  MoveL 652 to (-21.11, 309.47, 290) mm, rotated rx -90 ry -25 rz -110.46 deg; joints [2.992, -46.033, 98.025, 220.576, 108.57, -187.083, -1369.544]
  MoveL 653 to (-10.16, 196.36, 0) mm, rotated rx -90 ry -25 rz 39.27 deg; joints [-7.468, -49.927, 106.451, 214.616, 108.422, -179.076, -1519.273]
  Set speed (60.0 mm/s)
  MoveL 654 to (37.62, 209.05, 0) mm, rotated rx -90 ry -25 rz 92.57 deg; joints [-7.468, -49.977, 106.447, 214.605, 108.377, -179.109, -1572.574]
  MoveL 655 to (-10.16, 196.36, 0) mm, rotated rx -90 ry -25 rz 39.27 deg; joints [-7.468, -49.927, 106.451, 214.616, 108.422, -179.076, -1519.273]
  Set speed (60.0 mm/s)
  MoveL 656 to (-5.87, 195.78, 10) mm, rotated rx -90 ry -25 rz 43.82 deg; joints [-7.088, -49.822, 106.25, 214.856, 108.462, -179.315, -1523.823]
  MoveL 657 to (-1.12, 195.49, 20) mm, rotated rx -90 ry -25 rz 48.82 deg; joints [-6.709, -49.715, 106.043, 215.095, 108.501, -179.557, -1528.824]
  MoveL 658 to (4.03, 195.62, 30) mm, rotated rx -90 ry -25 rz 54.24 deg; joints [-6.332, -49.606, 105.829, 215.332, 108.536, -179.801, -1534.238]
  MoveL 659 to (9.5, 196.25, 40) mm, rotated rx -90 ry -25 rz 60.02 deg; joints [-5.956, -49.496, 105.609, 215.565, 108.567, -180.049, -1540.02]
  MoveL 660 to (15.19, 197.47, 50) mm, rotated rx -90 ry -25 rz 66.13 deg; joints [-5.581, -49.385, 105.383, 215.797, 108.596, -180.3, -1546.127]
  MoveL 661 to (21, 199.35, 60) mm, rotated rx -90 ry -25 rz 72.51 deg; joints [-5.207, -49.274, 105.15, 216.025, 108.62, -180.554, -1552.515]
  MoveL 662 to (26.8, 201.92, 70) mm, rotated rx -90 ry -25 rz 79.14 deg; joints [-4.834, -49.162, 104.91, 216.251, 108.64, -180.811, -1559.135]
  MoveL 663 to (32.46, 205.23, 80) mm, rotated rx -90 ry -25 rz 85.94 deg; joints [-4.463, -49.05, 104.664, 216.474, 108.657, -181.073, -1565.942]
  MoveL 664 to (37.86, 209.24, 90) mm, rotated rx -90 ry -25 rz 92.89 deg; joints [-4.093, -48.937, 104.412, 216.694, 108.67, -181.338, -1572.888]
  MoveL 665 to (42.85, 213.95, 100) mm, rotated rx -90 ry -25 rz 99.93 deg; joints [-3.725, -48.823, 104.153, 216.911, 108.679, -181.606, -1579.928]
  MoveL 666 to (47.33, 219.29, 110) mm, rotated rx -90 ry -25 rz 107.02 deg; joints [-3.358, -48.708, 103.888, 217.126, 108.685, -181.879, -1587.017]
  MoveL 667 to (51.17, 225.17, 120) mm, rotated rx -90 ry -25 rz 114.11 deg; joints [-2.992, -48.592, 103.616, 217.338, 108.687, -182.154, -1594.112]
  MoveL 668 to (54.3, 231.49, 130) mm, rotated rx -90 ry -25 rz 121.17 deg; joints [-2.628, -48.474, 103.338, 217.547, 108.687, -182.432, -1601.173]
  MoveL 669 to (56.65, 238.12, 140) mm, rotated rx -90 ry -25 rz 128.16 deg; joints [-2.265, -48.354, 103.054, 217.753, 108.685, -182.713, -1608.16]
  MoveL 670 to (58.18, 244.95, 150) mm, rotated rx -90 ry -25 rz 135.04 deg; joints [-1.904, -48.231, 102.763, 217.957, 108.681, -182.996, -1615.039]
  MoveL 671 to (58.89, 251.83, 160) mm, rotated rx -90 ry -25 rz 141.78 deg; joints [-1.544, -48.104, 102.465, 218.159, 108.676, -183.281, -1621.776]
  MoveL 672 to (58.8, 258.62, 170) mm, rotated rx -90 ry -25 rz 148.34 deg; joints [-1.185, -47.974, 102.162, 218.358, 108.669, -183.568, -1628.339]
  MoveL 673 to (57.96, 265.2, 180) mm, rotated rx -90 ry -25 rz 154.7 deg; joints [-0.828, -47.839, 101.852, 218.555, 108.662, -183.856, -1634.699]
  MoveL 674 to (56.44, 271.47, 190) mm, rotated rx -90 ry -25 rz 160.83 deg; joints [-0.473, -47.7, 101.535, 218.75, 108.655, -184.145, -1640.826]
  MoveL 675 to (54.33, 277.32, 200) mm, rotated rx -90 ry -25 rz 166.69 deg; joints [-0.119, -47.555, 101.213, 218.942, 108.647, -184.435, -1646.694]
  MoveL 676 to (51.74, 282.68, 210) mm, rotated rx -90 ry -25 rz 172.28 deg; joints [0.233, -47.406, 100.884, 219.133, 108.64, -184.725, -1652.275]
  MoveL 677 to (48.8, 287.5, 220) mm, rotated rx -90 ry -25 rz 177.54 deg; joints [0.584, -47.251, 100.549, 219.321, 108.632, -185.016, -1657.543]
  MoveL 678 to (45.62, 291.76, 230) mm, rotated rx -90 ry -25 rz -177.53 deg; joints [0.933, -47.091, 100.208, 219.507, 108.625, -185.308, -1662.471]
  MoveL 679 to (42.34, 295.45, 240) mm, rotated rx -90 ry -25 rz -172.97 deg; joints [1.28, -46.926, 99.86, 219.691, 108.618, -185.601, -1667.031]
  MoveL 680 to (39.07, 298.58, 250) mm, rotated rx -90 ry -25 rz -168.8 deg; joints [1.626, -46.755, 99.506, 219.873, 108.61, -185.894, -1671.197]
  MoveL 681 to (35.92, 301.18, 260) mm, rotated rx -90 ry -25 rz -165.06 deg; joints [1.97, -46.579, 99.146, 220.053, 108.603, -186.188, -1674.94]
  MoveL 682 to (33, 303.28, 270) mm, rotated rx -90 ry -25 rz -161.77 deg; joints [2.312, -46.398, 98.779, 220.231, 108.595, -186.483, -1678.23]
  MoveL 683 to (30.4, 304.94, 280) mm, rotated rx -90 ry -25 rz -158.96 deg; joints [2.653, -46.213, 98.406, 220.406, 108.587, -186.778, -1681.04]
  MoveL 684 to (28.22, 306.19, 290) mm, rotated rx -90 ry -25 rz -156.66 deg; joints [2.992, -46.023, 98.026, 220.579, 108.578, -187.075, -1683.337]
  MoveL 685 to (-21.11, 309.47, 290) mm, rotated rx -90 ry -25 rz -110.46 deg; joints [2.992, -46.033, 98.025, 220.576, 108.57, -187.083, -1729.544]
  Set speed (60.0 mm/s)
  MoveL 686 to (-18.74, 310.33, 280) mm, rotated rx -90 ry -25 rz -112.74 deg; joints [2.653, -46.23, 98.404, 220.402, 108.573, -186.791, -1727.257]
  MoveL 687 to (-15.8, 311.23, 270) mm, rotated rx -90 ry -25 rz -115.53 deg; joints [2.312, -46.424, 98.777, 220.225, 108.574, -186.502, -1724.467]
  MoveL 688 to (-12.3, 312.09, 260) mm, rotated rx -90 ry -25 rz -118.79 deg; joints [1.97, -46.614, 99.142, 220.045, 108.574, -186.214, -1721.209]
  MoveL 689 to (-8.28, 312.8, 250) mm, rotated rx -90 ry -25 rz -122.48 deg; joints [1.626, -46.801, 99.502, 219.863, 108.572, -185.928, -1717.515]
  MoveL 690 to (-3.78, 313.26, 240) mm, rotated rx -90 ry -25 rz -126.58 deg; joints [1.28, -46.983, 99.855, 219.678, 108.569, -185.643, -1713.419]
  MoveL 691 to (1.16, 313.37, 230) mm, rotated rx -90 ry -25 rz -131.05 deg; joints [0.933, -47.161, 100.201, 219.491, 108.565, -185.36, -1708.952]
  MoveL 692 to (6.46, 313.03, 220) mm, rotated rx -90 ry -25 rz -135.85 deg; joints [0.584, -47.335, 100.541, 219.301, 108.561, -185.078, -1704.147]
  MoveL 693 to (12.04, 312.14, 210) mm, rotated rx -90 ry -25 rz -140.97 deg; joints [0.233, -47.503, 100.875, 219.11, 108.557, -184.796, -1699.032]
  MoveL 694 to (17.8, 310.63, 200) mm, rotated rx -90 ry -25 rz -146.36 deg; joints [-0.119, -47.666, 101.203, 218.916, 108.553, -184.515, -1693.638]
  MoveL 695 to (23.62, 308.44, 190) mm, rotated rx -90 ry -25 rz -152.01 deg; joints [-0.473, -47.824, 101.524, 218.721, 108.549, -184.234, -1687.993]
  MoveL 696 to (29.38, 305.54, 180) mm, rotated rx -90 ry -25 rz -157.88 deg; joints [-0.828, -47.975, 101.839, 218.524, 108.546, -183.953, -1682.125]
  MoveL 697 to (34.94, 301.92, 170) mm, rotated rx -90 ry -25 rz -163.94 deg; joints [-1.185, -48.122, 102.148, 218.324, 108.543, -183.673, -1676.061]
  MoveL 698 to (40.17, 297.58, 160) mm, rotated rx -90 ry -25 rz -170.17 deg; joints [-1.544, -48.262, 102.451, 218.123, 108.54, -183.393, -1669.829]
  MoveL 699 to (44.94, 292.58, 150) mm, rotated rx -90 ry -25 rz -176.55 deg; joints [-1.904, -48.397, 102.748, 217.92, 108.539, -183.113, -1663.455]
  MoveL 700 to (49.15, 286.99, 140) mm, rotated rx -90 ry -25 rz 176.97 deg; joints [-2.265, -48.526, 103.038, 217.715, 108.537, -182.834, -1656.967]
  MoveL 701 to (52.68, 280.9, 130) mm, rotated rx -90 ry -25 rz 170.39 deg; joints [-2.628, -48.65, 103.323, 217.508, 108.536, -182.555, -1650.393]
  MoveL 702 to (55.46, 274.42, 120) mm, rotated rx -90 ry -25 rz 163.76 deg; joints [-2.992, -48.77, 103.601, 217.298, 108.534, -182.277, -1643.762]
  MoveL 703 to (57.44, 267.68, 110) mm, rotated rx -90 ry -25 rz 157.1 deg; joints [-3.358, -48.885, 103.873, 217.087, 108.532, -182, -1637.105]
  MoveL 704 to (58.6, 260.81, 100) mm, rotated rx -90 ry -25 rz 150.45 deg; joints [-3.725, -48.996, 104.139, 216.874, 108.529, -181.725, -1630.453]
  MoveL 705 to (58.95, 253.96, 90) mm, rotated rx -90 ry -25 rz 143.84 deg; joints [-4.093, -49.103, 104.398, 216.658, 108.525, -181.451, -1623.84]
  MoveL 706 to (58.51, 247.24, 80) mm, rotated rx -90 ry -25 rz 137.3 deg; joints [-4.463, -49.207, 104.652, 216.44, 108.52, -181.18, -1617.303]
  MoveL 707 to (57.35, 240.79, 70) mm, rotated rx -90 ry -25 rz 130.88 deg; joints [-4.834, -49.309, 104.898, 216.219, 108.512, -180.911, -1610.878]
  MoveL 708 to (55.55, 234.7, 60) mm, rotated rx -90 ry -25 rz 124.6 deg; joints [-5.207, -49.409, 105.139, 215.996, 108.502, -180.644, -1604.605]
  MoveL 709 to (53.21, 229.07, 50) mm, rotated rx -90 ry -25 rz 118.53 deg; joints [-5.581, -49.507, 105.373, 215.771, 108.489, -180.381, -1598.526]
  MoveL 710 to (50.45, 223.94, 40) mm, rotated rx -90 ry -25 rz 112.68 deg; joints [-5.956, -49.603, 105.601, 215.543, 108.473, -180.12, -1592.684]
  MoveL 711 to (47.39, 219.37, 30) mm, rotated rx -90 ry -25 rz 107.12 deg; joints [-6.332, -49.699, 105.822, 215.312, 108.454, -179.862, -1587.123]
  MoveL 712 to (44.15, 215.37, 20) mm, rotated rx -90 ry -25 rz 101.89 deg; joints [-6.709, -49.793, 106.037, 215.079, 108.432, -179.608, -1581.887]
  MoveL 713 to (40.85, 211.93, 10) mm, rotated rx -90 ry -25 rz 97.02 deg; joints [-7.088, -49.886, 106.245, 214.843, 108.406, -179.357, -1577.023]
  MoveL 714 to (37.62, 209.05, 0) mm, rotated rx -90 ry -25 rz 92.57 deg; joints [-7.468, -49.977, 106.447, 214.605, 108.377, -179.109, -1572.574]
  MoveL 715 to (-21.11, 309.47, 290) mm, rotated rx -90 ry -25 rz -110.46 deg; joints [2.992, -46.033, 98.025, 220.576, 108.57, -187.083, -1729.544]
  Set speed (60.0 mm/s)
  MoveL 716 to (-34.79, 325.15, 290) mm, rotated rx -90 ry -25 rz -105.16 deg; joints [2.992, -46.913, 97.922, 220.367, 107.822, -187.755, -1734.84]
  MoveL 717 to (37.62, 209.05, 0) mm, rotated rx -90 ry -25 rz 92.57 deg; joints [-7.468, -49.977, 106.447, 214.605, 108.377, -179.109, -1572.574]
  Set speed (60.0 mm/s)
  MoveL 718 to (55.59, 198.58, 0) mm, rotated rx -90 ry -25 rz 97.23 deg; joints [-7.468, -50.957, 106.353, 214.408, 107.492, -179.748, -1577.234]
  MoveL 719 to (37.62, 209.05, 0) mm, rotated rx -90 ry -25 rz 92.57 deg; joints [-7.468, -49.977, 106.447, 214.605, 108.377, -179.109, -1572.574]
  Set speed (60.0 mm/s)
  MoveL 720 to (40.85, 211.93, 10) mm, rotated rx -90 ry -25 rz 97.02 deg; joints [-7.088, -49.886, 106.245, 214.843, 108.406, -179.357, -1577.023]
  MoveL 721 to (44.15, 215.37, 20) mm, rotated rx -90 ry -25 rz 101.89 deg; joints [-6.709, -49.793, 106.037, 215.079, 108.432, -179.608, -1581.887]
  MoveL 722 to (47.39, 219.37, 30) mm, rotated rx -90 ry -25 rz 107.12 deg; joints [-6.332, -49.699, 105.822, 215.312, 108.454, -179.862, -1587.123]
  MoveL 723 to (50.45, 223.94, 40) mm, rotated rx -90 ry -25 rz 112.68 deg; joints [-5.956, -49.603, 105.601, 215.543, 108.473, -180.12, -1592.684]
  MoveL 724 to (53.21, 229.07, 50) mm, rotated rx -90 ry -25 rz 118.53 deg; joints [-5.581, -49.507, 105.373, 215.771, 108.489, -180.381, -1598.526]
  MoveL 725 to (55.55, 234.7, 60) mm, rotated rx -90 ry -25 rz 124.6 deg; joints [-5.207, -49.409, 105.139, 215.996, 108.502, -180.644, -1604.605]
  MoveL 726 to (57.35, 240.79, 70) mm, rotated rx -90 ry -25 rz 130.88 deg; joints [-4.834, -49.309, 104.898, 216.219, 108.512, -180.911, -1610.878]
  MoveL 727 to (58.51, 247.24, 80) mm, rotated rx -90 ry -25 rz 137.3 deg; joints [-4.463, -49.207, 104.652, 216.44, 108.52, -181.18, -1617.303]
  MoveL 728 to (58.95, 253.96, 90) mm, rotated rx -90 ry -25 rz 143.84 deg; joints [-4.093, -49.103, 104.398, 216.658, 108.525, -181.451, -1623.84]
  MoveL 729 to (58.6, 260.81, 100) mm, rotated rx -90 ry -25 rz 150.45 deg; joints [-3.725, -48.996, 104.139, 216.874, 108.529, -181.725, -1630.453]
  MoveL 730 to (57.44, 267.68, 110) mm, rotated rx -90 ry -25 rz 157.1 deg; joints [-3.358, -48.885, 103.873, 217.087, 108.532, -182, -1637.105]
  MoveL 731 to (55.46, 274.42, 120) mm, rotated rx -90 ry -25 rz 163.76 deg; joints [-2.992, -48.77, 103.601, 217.298, 108.534, -182.277, -1643.762]
  MoveL 732 to (52.68, 280.9, 130) mm, rotated rx -90 ry -25 rz 170.39 deg; joints [-2.628, -48.65, 103.323, 217.508, 108.536, -182.555, -1650.393]
  MoveL 733 to (49.15, 286.99, 140) mm, rotated rx -90 ry -25 rz 176.97 deg; joints [-2.265, -48.526, 103.038, 217.715, 108.537, -182.834, -1656.967]
  MoveL 734 to (44.94, 292.58, 150) mm, rotated rx -90 ry -25 rz -176.55 deg; joints [-1.904, -48.397, 102.748, 217.92, 108.539, -183.113, -1663.455]
  MoveL 735 to (40.17, 297.58, 160) mm, rotated rx -90 ry -25 rz -170.17 deg; joints [-1.544, -48.262, 102.451, 218.123, 108.54, -183.393, -1669.829]
  MoveL 736 to (34.94, 301.92, 170) mm, rotated rx -90 ry -25 rz -163.94 deg; joints [-1.185, -48.122, 102.148, 218.324, 108.543, -183.673, -1676.061]
  MoveL 737 to (29.38, 305.54, 180) mm, rotated rx -90 ry -25 rz -157.88 deg; joints [-0.828, -47.975, 101.839, 218.524, 108.546, -183.953, -1682.125]
  MoveL 738 to (23.62, 308.44, 190) mm, rotated rx -90 ry -25 rz -152.01 deg; joints [-0.473, -47.824, 101.524, 218.721, 108.549, -184.234, -1687.993]
  MoveL 739 to (17.8, 310.63, 200) mm, rotated rx -90 ry -25 rz -146.36 deg; joints [-0.119, -47.666, 101.203, 218.916, 108.553, -184.515, -1693.638]
  MoveL 740 to (12.04, 312.14, 210) mm, rotated rx -90 ry -25 rz -140.97 deg; joints [0.233, -47.503, 100.875, 219.11, 108.557, -184.796, -1699.032]
  MoveL 741 to (6.46, 313.03, 220) mm, rotated rx -90 ry -25 rz -135.85 deg; joints [0.584, -47.335, 100.541, 219.301, 108.561, -185.078, -1704.147]
  MoveL 742 to (1.16, 313.37, 230) mm, rotated rx -90 ry -25 rz -131.05 deg; joints [0.933, -47.161, 100.201, 219.491, 108.565, -185.36, -1708.952]
  MoveL 743 to (-3.78, 313.26, 240) mm, rotated rx -90 ry -25 rz -126.58 deg; joints [1.28, -46.983, 99.855, 219.678, 108.569, -185.643, -1713.419]
  MoveL 744 to (-8.28, 312.8, 250) mm, rotated rx -90 ry -25 rz -122.48 deg; joints [1.626, -46.801, 99.502, 219.863, 108.572, -185.928, -1717.515]
  MoveL 745 to (-12.3, 312.09, 260) mm, rotated rx -90 ry -25 rz -118.79 deg; joints [1.97, -46.614, 99.142, 220.045, 108.574, -186.214, -1721.209]
  MoveL 746 to (-15.8, 311.23, 270) mm, rotated rx -90 ry -25 rz -115.53 deg; joints [2.312, -46.424, 98.777, 220.225, 108.574, -186.502, -1724.467]
  MoveL 747 to (-18.74, 310.33, 280) mm, rotated rx -90 ry -25 rz -112.74 deg; joints [2.653, -46.23, 98.404, 220.402, 108.573, -186.791, -1727.257]
  MoveL 748 to (-21.11, 309.47, 290) mm, rotated rx -90 ry -25 rz -110.46 deg; joints [2.992, -46.033, 98.025, 220.576, 108.57, -187.083, -1729.544]
  MoveL 749 to (-34.79, 325.15, 290) mm, rotated rx -90 ry -25 rz -105.16 deg; joints [2.992, -46.913, 97.922, 220.367, 107.822, -187.755, -1734.84]
  Set speed (60.0 mm/s)
  MoveL 750 to (-31.73, 326.57, 280) mm, rotated rx -90 ry -25 rz -107.49 deg; joints [2.653, -47.114, 98.301, 220.192, 107.82, -187.463, -1732.51]
  MoveL 751 to (-27.92, 328.13, 270) mm, rotated rx -90 ry -25 rz -110.33 deg; joints [2.312, -47.311, 98.673, 220.015, 107.816, -187.174, -1729.668]
  MoveL 752 to (-23.38, 329.69, 260) mm, rotated rx -90 ry -25 rz -113.65 deg; joints [1.97, -47.505, 99.038, 219.835, 107.811, -186.886, -1726.348]
  MoveL 753 to (-18.11, 331.13, 250) mm, rotated rx -90 ry -25 rz -117.42 deg; joints [1.626, -47.696, 99.397, 219.652, 107.803, -186.601, -1722.585]
  MoveL 754 to (-12.17, 332.29, 240) mm, rotated rx -90 ry -25 rz -121.59 deg; joints [1.28, -47.883, 99.75, 219.468, 107.795, -186.317, -1718.413]
  MoveL 755 to (-5.61, 333.04, 230) mm, rotated rx -90 ry -25 rz -126.13 deg; joints [0.933, -48.065, 100.096, 219.281, 107.786, -186.034, -1713.865]
  MoveL 756 to (1.49, 333.22, 220) mm, rotated rx -90 ry -25 rz -131.03 deg; joints [0.584, -48.243, 100.436, 219.091, 107.776, -185.752, -1708.974]
  MoveL 757 to (9.03, 332.72, 210) mm, rotated rx -90 ry -25 rz -136.23 deg; joints [0.233, -48.416, 100.77, 218.9, 107.766, -185.47, -1703.771]
  MoveL 758 to (16.88, 331.41, 200) mm, rotated rx -90 ry -25 rz -141.71 deg; joints [-0.119, -48.583, 101.097, 218.706, 107.756, -185.189, -1698.287]
  MoveL 759 to (24.89, 329.2, 190) mm, rotated rx -90 ry -25 rz -147.45 deg; joints [-0.473, -48.745, 101.419, 218.511, 107.747, -184.908, -1692.553]
  MoveL 760 to (32.91, 326.04, 180) mm, rotated rx -90 ry -25 rz -153.4 deg; joints [-0.828, -48.902, 101.734, 218.314, 107.738, -184.628, -1686.599]
  MoveL 761 to (40.75, 321.89, 170) mm, rotated rx -90 ry -25 rz -159.55 deg; joints [-1.185, -49.052, 102.043, 218.114, 107.729, -184.347, -1680.453]
  MoveL 762 to (48.24, 316.75, 160) mm, rotated rx -90 ry -25 rz -165.85 deg; joints [-1.544, -49.197, 102.347, 217.913, 107.721, -184.067, -1674.145]
  MoveL 763 to (55.2, 310.67, 150) mm, rotated rx -90 ry -25 rz -172.3 deg; joints [-1.904, -49.336, 102.644, 217.71, 107.714, -183.786, -1667.704]
  MoveL 764 to (61.48, 303.74, 140) mm, rotated rx -90 ry -25 rz -178.84 deg; joints [-2.265, -49.47, 102.935, 217.505, 107.707, -183.506, -1661.158]
  MoveL 765 to (66.92, 296.06, 130) mm, rotated rx -90 ry -25 rz 174.54 deg; joints [-2.628, -49.598, 103.22, 217.299, 107.701, -183.226, -1654.539]
  MoveL 766 to (71.41, 287.77, 120) mm, rotated rx -90 ry -25 rz 167.87 deg; joints [-2.992, -49.721, 103.499, 217.09, 107.695, -182.947, -1647.875]
  MoveL 767 to (74.87, 279.04, 110) mm, rotated rx -90 ry -25 rz 161.2 deg; joints [-3.358, -49.84, 103.771, 216.879, 107.688, -182.669, -1641.198]
  MoveL 768 to (77.24, 270.04, 100) mm, rotated rx -90 ry -25 rz 154.54 deg; joints [-3.725, -49.954, 104.038, 216.666, 107.681, -182.392, -1634.542]
  MoveL 769 to (78.53, 260.95, 90) mm, rotated rx -90 ry -25 rz 147.94 deg; joints [-4.093, -50.065, 104.298, 216.451, 107.672, -182.117, -1627.94]
  MoveL 770 to (78.77, 251.96, 80) mm, rotated rx -90 ry -25 rz 141.43 deg; joints [-4.463, -50.172, 104.552, 216.234, 107.663, -181.843, -1621.427]
  MoveL 771 to (78, 243.23, 70) mm, rotated rx -90 ry -25 rz 135.04 deg; joints [-4.834, -50.277, 104.8, 216.014, 107.651, -181.572, -1615.041]
  MoveL 772 to (76.35, 234.91, 60) mm, rotated rx -90 ry -25 rz 128.82 deg; joints [-5.207, -50.379, 105.041, 215.792, 107.637, -181.303, -1608.819]
  MoveL 773 to (73.92, 227.12, 50) mm, rotated rx -90 ry -25 rz 122.8 deg; joints [-5.581, -50.479, 105.276, 215.568, 107.62, -181.036, -1602.802]
  MoveL 774 to (70.87, 219.96, 40) mm, rotated rx -90 ry -25 rz 117.03 deg; joints [-5.956, -50.577, 105.504, 215.341, 107.601, -180.773, -1597.03]
  MoveL 775 to (67.34, 213.5, 30) mm, rotated rx -90 ry -25 rz 111.55 deg; joints [-6.332, -50.674, 105.726, 215.111, 107.579, -180.512, -1591.545]
  MoveL 776 to (63.51, 207.78, 20) mm, rotated rx -90 ry -25 rz 106.39 deg; joints [-6.709, -50.77, 105.941, 214.879, 107.553, -180.254, -1586.389]
  MoveL 777 to (59.54, 202.81, 10) mm, rotated rx -90 ry -25 rz 101.6 deg; joints [-7.088, -50.864, 106.15, 214.645, 107.524, -180, -1581.605]
  MoveL 778 to (55.59, 198.58, 0) mm, rotated rx -90 ry -25 rz 97.23 deg; joints [-7.468, -50.957, 106.353, 214.408, 107.492, -179.748, -1577.234]
  MoveL 779 to (-34.79, 325.15, 290) mm, rotated rx -90 ry -25 rz -105.16 deg; joints [2.992, -46.913, 97.922, 220.367, 107.822, -187.755, -1734.84]
  Set speed (60.0 mm/s)
  MoveL 780 to (-30.72, 304.75, 290) mm, rotated rx -90 ry -25 rz -100.71 deg; joints [2.992, -46.018, 98.027, 220.58, 108.582, -187.072, -1739.294]
  MoveL 781 to (55.59, 198.58, 0) mm, rotated rx -90 ry -25 rz 97.23 deg; joints [-7.468, -50.957, 106.353, 214.408, 107.492, -179.748, -1577.234]
  Set speed (60.0 mm/s)
  MoveL 782 to (45.21, 216.6, 0) mm, rotated rx -90 ry -25 rz 103.54 deg; joints [-7.468, -50.007, 106.445, 214.599, 108.351, -179.128, -1583.543]
  MoveL 783 to (55.59, 198.58, 0) mm, rotated rx -90 ry -25 rz 97.23 deg; joints [-7.468, -50.957, 106.353, 214.408, 107.492, -179.748, -1577.234]
  Set speed (60.0 mm/s)
  MoveL 784 to (59.54, 202.81, 10) mm, rotated rx -90 ry -25 rz 101.6 deg; joints [-7.088, -50.864, 106.15, 214.645, 107.524, -180, -1581.605]
  MoveL 785 to (63.51, 207.78, 20) mm, rotated rx -90 ry -25 rz 106.39 deg; joints [-6.709, -50.77, 105.941, 214.879, 107.553, -180.254, -1586.389]
  MoveL 786 to (67.34, 213.5, 30) mm, rotated rx -90 ry -25 rz 111.55 deg; joints [-6.332, -50.674, 105.726, 215.111, 107.579, -180.512, -1591.545]
  MoveL 787 to (70.87, 219.96, 40) mm, rotated rx -90 ry -25 rz 117.03 deg; joints [-5.956, -50.577, 105.504, 215.341, 107.601, -180.773, -1597.03]
  MoveL 788 to (73.92, 227.12, 50) mm, rotated rx -90 ry -25 rz 122.8 deg; joints [-5.581, -50.479, 105.276, 215.568, 107.62, -181.036, -1602.802]
  MoveL 789 to (76.35, 234.91, 60) mm, rotated rx -90 ry -25 rz 128.82 deg; joints [-5.207, -50.379, 105.041, 215.792, 107.637, -181.303, -1608.819]
  MoveL 790 to (78, 243.23, 70) mm, rotated rx -90 ry -25 rz 135.04 deg; joints [-4.834, -50.277, 104.8, 216.014, 107.651, -181.572, -1615.041]
  MoveL 791 to (78.77, 251.96, 80) mm, rotated rx -90 ry -25 rz 141.43 deg; joints [-4.463, -50.172, 104.552, 216.234, 107.663, -181.843, -1621.427]
  MoveL 792 to (78.53, 260.95, 90) mm, rotated rx -90 ry -25 rz 147.94 deg; joints [-4.093, -50.065, 104.298, 216.451, 107.672, -182.117, -1627.94]
  MoveL 793 to (77.24, 270.04, 100) mm, rotated rx -90 ry -25 rz 154.54 deg; joints [-3.725, -49.954, 104.038, 216.666, 107.681, -182.392, -1634.542]
  MoveL 794 to (74.87, 279.04, 110) mm, rotated rx -90 ry -25 rz 161.2 deg; joints [-3.358, -49.84, 103.771, 216.879, 107.688, -182.669, -1641.198]
  MoveL 795 to (71.41, 287.77, 120) mm, rotated rx -90 ry -25 rz 167.87 deg; joints [-2.992, -49.721, 103.499, 217.09, 107.695, -182.947, -1647.875]
  MoveL 796 to (66.92, 296.06, 130) mm, rotated rx -90 ry -25 rz 174.54 deg; joints [-2.628, -49.598, 103.22, 217.299, 107.701, -183.226, -1654.539]
  MoveL 797 to (61.48, 303.74, 140) mm, rotated rx -90 ry -25 rz -178.84 deg; joints [-2.265, -49.47, 102.935, 217.505, 107.707, -183.506, -1661.158]
  MoveL 798 to (55.2, 310.67, 150) mm, rotated rx -90 ry -25 rz -172.3 deg; joints [-1.904, -49.336, 102.644, 217.71, 107.714, -183.786, -1667.704]
  MoveL 799 to (48.24, 316.75, 160) mm, rotated rx -90 ry -25 rz -165.85 deg; joints [-1.544, -49.197, 102.347, 217.913, 107.721, -184.067, -1674.145]
  MoveL 800 to (40.75, 321.89, 170) mm, rotated rx -90 ry -25 rz -159.55 deg; joints [-1.185, -49.052, 102.043, 218.114, 107.729, -184.347, -1680.453]
  MoveL 801 to (32.91, 326.04, 180) mm, rotated rx -90 ry -25 rz -153.4 deg; joints [-0.828, -48.902, 101.734, 218.314, 107.738, -184.628, -1686.599]
  MoveL 802 to (24.89, 329.2, 190) mm, rotated rx -90 ry -25 rz -147.45 deg; joints [-0.473, -48.745, 101.419, 218.511, 107.747, -184.908, -1692.553]
  MoveL 803 to (16.88, 331.41, 200) mm, rotated rx -90 ry -25 rz -141.71 deg; joints [-0.119, -48.583, 101.097, 218.706, 107.756, -185.189, -1698.287]
  MoveL 804 to (9.03, 332.72, 210) mm, rotated rx -90 ry -25 rz -136.23 deg; joints [0.233, -48.416, 100.77, 218.9, 107.766, -185.47, -1703.771]
  MoveL 805 to (1.49, 333.22, 220) mm, rotated rx -90 ry -25 rz -131.03 deg; joints [0.584, -48.243, 100.436, 219.091, 107.776, -185.752, -1708.974]
  MoveL 806 to (-5.61, 333.04, 230) mm, rotated rx -90 ry -25 rz -126.13 deg; joints [0.933, -48.065, 100.096, 219.281, 107.786, -186.034, -1713.865]
  MoveL 807 to (-12.17, 332.29, 240) mm, rotated rx -90 ry -25 rz -121.59 deg; joints [1.28, -47.883, 99.75, 219.468, 107.795, -186.317, -1718.413]
  MoveL 808 to (-18.11, 331.13, 250) mm, rotated rx -90 ry -25 rz -117.42 deg; joints [1.626, -47.696, 99.397, 219.652, 107.803, -186.601, -1722.585]
  MoveL 809 to (-23.38, 329.69, 260) mm, rotated rx -90 ry -25 rz -113.65 deg; joints [1.97, -47.505, 99.038, 219.835, 107.811, -186.886, -1726.348]
  MoveL 810 to (-27.92, 328.13, 270) mm, rotated rx -90 ry -25 rz -110.33 deg; joints [2.312, -47.311, 98.673, 220.015, 107.816, -187.174, -1729.668]
  MoveL 811 to (-31.73, 326.57, 280) mm, rotated rx -90 ry -25 rz -107.49 deg; joints [2.653, -47.114, 98.301, 220.192, 107.82, -187.463, -1732.51]
  MoveL 812 to (-34.79, 325.15, 290) mm, rotated rx -90 ry -25 rz -105.16 deg; joints [2.992, -46.913, 97.922, 220.367, 107.822, -187.755, -1734.84]
  MoveL 813 to (-30.72, 304.75, 290) mm, rotated rx -90 ry -25 rz -100.71 deg; joints [2.992, -46.018, 98.027, 220.58, 108.582, -187.072, -1739.294]
  Set speed (60.0 mm/s)
  MoveL 814 to (-28.54, 306.02, 280) mm, rotated rx -90 ry -25 rz -103 deg; joints [2.653, -46.216, 98.406, 220.405, 108.584, -186.781, -1736.997]
  MoveL 815 to (-25.81, 307.44, 270) mm, rotated rx -90 ry -25 rz -105.8 deg; joints [2.312, -46.412, 98.778, 220.228, 108.584, -186.493, -1734.195]
  MoveL 816 to (-22.53, 308.91, 260) mm, rotated rx -90 ry -25 rz -109.08 deg; joints [1.97, -46.604, 99.143, 220.047, 108.582, -186.206, -1730.925]
  MoveL 817 to (-18.7, 310.34, 250) mm, rotated rx -90 ry -25 rz -112.78 deg; joints [1.626, -46.793, 99.502, 219.864, 108.579, -185.922, -1727.22]
  MoveL 818 to (-14.35, 311.61, 240) mm, rotated rx -90 ry -25 rz -116.88 deg; joints [1.28, -46.978, 99.855, 219.679, 108.574, -185.639, -1723.116]
  MoveL 819 to (-9.52, 312.61, 230) mm, rotated rx -90 ry -25 rz -121.36 deg; joints [0.933, -47.159, 100.201, 219.491, 108.568, -185.358, -1718.643]
  MoveL 820 to (-4.24, 313.23, 220) mm, rotated rx -90 ry -25 rz -126.16 deg; joints [0.584, -47.335, 100.541, 219.301, 108.561, -185.078, -1713.836]
  MoveL 821 to (1.41, 313.37, 210) mm, rotated rx -90 ry -25 rz -131.27 deg; joints [0.233, -47.507, 100.875, 219.109, 108.554, -184.799, -1708.726]
  MoveL 822 to (7.35, 312.92, 200) mm, rotated rx -90 ry -25 rz -136.66 deg; joints [-0.119, -47.673, 101.202, 218.915, 108.547, -184.52, -1703.341]
  MoveL 823 to (13.47, 311.83, 190) mm, rotated rx -90 ry -25 rz -142.29 deg; joints [-0.473, -47.835, 101.523, 218.718, 108.54, -184.242, -1697.713]
  MoveL 824 to (19.65, 310.01, 180) mm, rotated rx -90 ry -25 rz -148.13 deg; joints [-0.828, -47.99, 101.838, 218.52, 108.533, -183.964, -1691.868]
  MoveL 825 to (25.78, 307.45, 170) mm, rotated rx -90 ry -25 rz -154.16 deg; joints [-1.185, -48.14, 102.146, 218.32, 108.527, -183.686, -1685.836]
  MoveL 826 to (31.7, 304.13, 160) mm, rotated rx -90 ry -25 rz -160.36 deg; joints [-1.544, -48.284, 102.449, 218.118, 108.522, -183.409, -1679.644]
  MoveL 827 to (37.3, 300.08, 150) mm, rotated rx -90 ry -25 rz -166.68 deg; joints [-1.904, -48.422, 102.745, 217.914, 108.517, -183.131, -1673.318]
  MoveL 828 to (42.45, 295.34, 140) mm, rotated rx -90 ry -25 rz -173.11 deg; joints [-2.265, -48.554, 103.036, 217.708, 108.513, -182.854, -1666.886]
  MoveL 829 to (47.02, 289.99, 130) mm, rotated rx -90 ry -25 rz -179.62 deg; joints [-2.628, -48.681, 103.32, 217.501, 108.509, -182.577, -1660.375]
  MoveL 830 to (50.93, 284.12, 120) mm, rotated rx -90 ry -25 rz 173.82 deg; joints [-2.992, -48.803, 103.598, 217.291, 108.505, -182.3, -1653.815]
  MoveL 831 to (54.1, 277.85, 110) mm, rotated rx -90 ry -25 rz 167.23 deg; joints [-3.358, -48.92, 103.87, 217.079, 108.501, -182.025, -1647.235]
  MoveL 832 to (56.49, 271.3, 100) mm, rotated rx -90 ry -25 rz 160.66 deg; joints [-3.725, -49.033, 104.136, 216.866, 108.497, -181.75, -1640.664]
  MoveL 833 to (58.06, 264.62, 90) mm, rotated rx -90 ry -25 rz 154.14 deg; joints [-4.093, -49.141, 104.395, 216.65, 108.492, -181.477, -1634.137]
  MoveL 834 to (58.85, 257.94, 80) mm, rotated rx -90 ry -25 rz 147.69 deg; joints [-4.463, -49.246, 104.648, 216.431, 108.486, -181.206, -1627.686]
  MoveL 835 to (58.87, 251.39, 70) mm, rotated rx -90 ry -25 rz 141.35 deg; joints [-4.834, -49.348, 104.895, 216.211, 108.478, -180.937, -1621.348]
  MoveL 836 to (58.2, 245.07, 60) mm, rotated rx -90 ry -25 rz 135.16 deg; joints [-5.207, -49.447, 105.136, 215.988, 108.468, -180.67, -1615.162]
  MoveL 837 to (56.92, 239.11, 50) mm, rotated rx -90 ry -25 rz 129.17 deg; joints [-5.581, -49.545, 105.37, 215.763, 108.456, -180.406, -1609.166]
  MoveL 838 to (55.13, 233.57, 40) mm, rotated rx -90 ry -25 rz 123.4 deg; joints [-5.956, -49.64, 105.598, 215.535, 108.441, -180.144, -1603.403]
  MoveL 839 to (52.95, 228.52, 30) mm, rotated rx -90 ry -25 rz 117.91 deg; joints [-6.332, -49.733, 105.819, 215.305, 108.423, -179.885, -1597.915]
  MoveL 840 to (50.48, 223.99, 20) mm, rotated rx -90 ry -25 rz 112.75 deg; joints [-6.709, -49.826, 106.034, 215.072, 108.402, -179.63, -1592.746]
  MoveL 841 to (47.86, 220.02, 10) mm, rotated rx -90 ry -25 rz 107.94 deg; joints [-7.088, -49.917, 106.243, 214.837, 108.378, -179.377, -1587.94]
  MoveL 842 to (45.21, 216.6, 0) mm, rotated rx -90 ry -25 rz 103.54 deg; joints [-7.468, -50.007, 106.445, 214.599, 108.351, -179.128, -1583.543]
  MoveL 843 to (-30.72, 304.75, 290) mm, rotated rx -90 ry -25 rz -100.71 deg; joints [2.992, -46.018, 98.027, 220.58, 108.582, -187.072, -1739.294]
  Set speed (60.0 mm/s)
  MoveL 844 to (-58.22, 263.67, 290) mm, rotated rx -90 ry -25 rz -53.21 deg; joints [2.992, -45.884, 98.039, 220.612, 108.694, -186.971, -1786.787]
  MoveL 845 to (45.21, 216.6, 0) mm, rotated rx -90 ry -25 rz 103.54 deg; joints [-7.468, -50.007, 106.445, 214.599, 108.351, -179.128, -1943.543]
  Set speed (60.0 mm/s)
  MoveL 846 to (58.12, 264.32, 0) mm, rotated rx -90 ry -25 rz 153.85 deg; joints [-7.468, -50.186, 106.43, 214.563, 108.191, -179.243, -1993.845]
  MoveL 847 to (45.21, 216.6, 0) mm, rotated rx -90 ry -25 rz 103.54 deg; joints [-7.468, -50.007, 106.445, 214.599, 108.351, -179.128, -1943.543]
  Set speed (60.0 mm/s)
  MoveL 848 to (47.86, 220.02, 10) mm, rotated rx -90 ry -25 rz 107.94 deg; joints [-7.088, -49.917, 106.243, 214.837, 108.378, -179.377, -1947.94]
  MoveL 849 to (50.48, 223.99, 20) mm, rotated rx -90 ry -25 rz 112.75 deg; joints [-6.709, -49.826, 106.034, 215.072, 108.402, -179.63, -1952.746]
  MoveL 850 to (52.95, 228.52, 30) mm, rotated rx -90 ry -25 rz 117.91 deg; joints [-6.332, -49.733, 105.819, 215.305, 108.423, -179.885, -1957.915]
  MoveL 851 to (55.13, 233.57, 40) mm, rotated rx -90 ry -25 rz 123.4 deg; joints [-5.956, -49.64, 105.598, 215.535, 108.441, -180.144, -1963.403]
  MoveL 852 to (56.92, 239.11, 50) mm, rotated rx -90 ry -25 rz 129.17 deg; joints [-5.581, -49.545, 105.37, 215.763, 108.456, -180.406, -1969.166]
  MoveL 853 to (58.2, 245.07, 60) mm, rotated rx -90 ry -25 rz 135.16 deg; joints [-5.207, -49.447, 105.136, 215.988, 108.468, -180.67, -1975.162]
  MoveL 854 to (58.87, 251.39, 70) mm, rotated rx -90 ry -25 rz 141.35 deg; joints [-4.834, -49.348, 104.895, 216.211, 108.478, -180.937, -1981.348]
  MoveL 855 to (58.85, 257.94, 80) mm, rotated rx -90 ry -25 rz 147.69 deg; joints [-4.463, -49.246, 104.648, 216.431, 108.486, -181.206, -1987.686]
  MoveL 856 to (58.06, 264.62, 90) mm, rotated rx -90 ry -25 rz 154.14 deg; joints [-4.093, -49.141, 104.395, 216.65, 108.492, -181.477, -1994.137]
  MoveL 857 to (56.49, 271.3, 100) mm, rotated rx -90 ry -25 rz 160.66 deg; joints [-3.725, -49.033, 104.136, 216.866, 108.497, -181.75, -2000.664]
  MoveL 858 to (54.1, 277.85, 110) mm, rotated rx -90 ry -25 rz 167.23 deg; joints [-3.358, -48.92, 103.87, 217.079, 108.501, -182.025, -2007.235]
  MoveL 859 to (50.93, 284.12, 120) mm, rotated rx -90 ry -25 rz 173.82 deg; joints [-2.992, -48.803, 103.598, 217.291, 108.505, -182.3, -2013.815]
  MoveL 860 to (47.02, 289.99, 130) mm, rotated rx -90 ry -25 rz -179.62 deg; joints [-2.628, -48.681, 103.32, 217.501, 108.509, -182.577, -2020.375]
  MoveL 861 to (42.45, 295.34, 140) mm, rotated rx -90 ry -25 rz -173.11 deg; joints [-2.265, -48.554, 103.036, 217.708, 108.513, -182.854, -2026.886]
  MoveL 862 to (37.3, 300.08, 150) mm, rotated rx -90 ry -25 rz -166.68 deg; joints [-1.904, -48.422, 102.745, 217.914, 108.517, -183.131, -2033.318]
  MoveL 863 to (31.7, 304.13, 160) mm, rotated rx -90 ry -25 rz -160.36 deg; joints [-1.544, -48.284, 102.449, 218.118, 108.522, -183.409, -2039.644]
  MoveL 864 to (25.78, 307.45, 170) mm, rotated rx -90 ry -25 rz -154.16 deg; joints [-1.185, -48.14, 102.146, 218.32, 108.527, -183.686, -2045.836]
  MoveL 865 to (19.65, 310.01, 180) mm, rotated rx -90 ry -25 rz -148.13 deg; joints [-0.828, -47.99, 101.838, 218.52, 108.533, -183.964, -2051.868]
  MoveL 866 to (13.47, 311.83, 190) mm, rotated rx -90 ry -25 rz -142.29 deg; joints [-0.473, -47.835, 101.523, 218.718, 108.54, -184.242, -2057.713]
  MoveL 867 to (7.35, 312.92, 200) mm, rotated rx -90 ry -25 rz -136.66 deg; joints [-0.119, -47.673, 101.202, 218.915, 108.547, -184.52, -2063.341]
  MoveL 868 to (1.41, 313.37, 210) mm, rotated rx -90 ry -25 rz -131.27 deg; joints [0.233, -47.507, 100.875, 219.109, 108.554, -184.799, -2068.726]
  MoveL 869 to (-4.24, 313.23, 220) mm, rotated rx -90 ry -25 rz -126.16 deg; joints [0.584, -47.335, 100.541, 219.301, 108.561, -185.078, -2073.836]
  MoveL 870 to (-9.52, 312.61, 230) mm, rotated rx -90 ry -25 rz -121.36 deg; joints [0.933, -47.159, 100.201, 219.491, 108.568, -185.358, -2078.643]
  MoveL 871 to (-14.35, 311.61, 240) mm, rotated rx -90 ry -25 rz -116.88 deg; joints [1.28, -46.978, 99.855, 219.679, 108.574, -185.639, -2083.116]
  MoveL 872 to (-18.7, 310.34, 250) mm, rotated rx -90 ry -25 rz -112.78 deg; joints [1.626, -46.793, 99.502, 219.864, 108.579, -185.922, -2087.22]
  MoveL 873 to (-22.53, 308.91, 260) mm, rotated rx -90 ry -25 rz -109.08 deg; joints [1.97, -46.604, 99.143, 220.047, 108.582, -186.206, -2090.925]
  MoveL 874 to (-25.81, 307.44, 270) mm, rotated rx -90 ry -25 rz -105.8 deg; joints [2.312, -46.412, 98.778, 220.228, 108.584, -186.493, -2094.195]
  MoveL 875 to (-28.54, 306.02, 280) mm, rotated rx -90 ry -25 rz -103 deg; joints [2.653, -46.216, 98.406, 220.405, 108.584, -186.781, -2096.997]
  MoveL 876 to (-30.72, 304.75, 290) mm, rotated rx -90 ry -25 rz -100.71 deg; joints [2.992, -46.018, 98.027, 220.58, 108.582, -187.072, -2099.294]
  MoveL 877 to (-58.22, 263.67, 290) mm, rotated rx -90 ry -25 rz -53.21 deg; joints [2.992, -45.884, 98.039, 220.612, 108.694, -186.971, -2146.787]
  Set speed (60.0 mm/s)
  MoveL 878 to (-57.77, 266.15, 280) mm, rotated rx -90 ry -25 rz -55.62 deg; joints [2.653, -46.086, 98.418, 220.436, 108.693, -186.683, -2144.382]
  MoveL 879 to (-57.08, 269.15, 270) mm, rotated rx -90 ry -25 rz -58.54 deg; joints [2.312, -46.286, 98.79, 220.257, 108.689, -186.399, -2141.455]
  MoveL 880 to (-56.08, 272.6, 260) mm, rotated rx -90 ry -25 rz -61.95 deg; joints [1.97, -46.485, 99.155, 220.076, 108.682, -186.118, -2138.047]
  MoveL 881 to (-54.69, 276.44, 250) mm, rotated rx -90 ry -25 rz -65.8 deg; joints [1.626, -46.682, 99.513, 219.891, 108.672, -185.84, -2134.197]
  MoveL 882 to (-52.84, 280.57, 240) mm, rotated rx -90 ry -25 rz -70.06 deg; joints [1.28, -46.876, 99.865, 219.703, 108.659, -185.564, -2129.944]
  MoveL 883 to (-50.46, 284.91, 230) mm, rotated rx -90 ry -25 rz -74.67 deg; joints [0.933, -47.068, 100.21, 219.513, 108.644, -185.292, -2125.328]
  MoveL 884 to (-47.51, 289.33, 220) mm, rotated rx -90 ry -25 rz -79.61 deg; joints [0.584, -47.257, 100.549, 219.32, 108.627, -185.021, -2120.386]
  MoveL 885 to (-43.95, 293.72, 210) mm, rotated rx -90 ry -25 rz -84.84 deg; joints [0.233, -47.443, 100.881, 219.124, 108.608, -184.752, -2115.156]
  MoveL 886 to (-39.77, 297.95, 200) mm, rotated rx -90 ry -25 rz -90.33 deg; joints [-0.119, -47.624, 101.206, 218.926, 108.588, -184.485, -2109.672]
  MoveL 887 to (-34.96, 301.9, 190) mm, rotated rx -90 ry -25 rz -96.03 deg; joints [-0.473, -47.802, 101.526, 218.726, 108.567, -184.218, -2103.97]
  MoveL 888 to (-29.57, 305.43, 180) mm, rotated rx -90 ry -25 rz -101.92 deg; joints [-0.828, -47.975, 101.839, 218.524, 108.546, -183.953, -2098.081]
  MoveL 889 to (-23.65, 308.43, 170) mm, rotated rx -90 ry -25 rz -107.96 deg; joints [-1.185, -48.143, 102.146, 218.319, 108.524, -183.689, -2092.038]
  MoveL 890 to (-17.28, 310.79, 160) mm, rotated rx -90 ry -25 rz -114.13 deg; joints [-1.544, -48.306, 102.447, 218.113, 108.503, -183.424, -2085.87]
  MoveL 891 to (-10.57, 312.43, 150) mm, rotated rx -90 ry -25 rz -120.39 deg; joints [-1.904, -48.463, 102.742, 217.905, 108.481, -183.16, -2079.606]
  MoveL 892 to (-3.62, 313.27, 140) mm, rotated rx -90 ry -25 rz -126.72 deg; joints [-2.265, -48.614, 103.03, 217.695, 108.461, -182.896, -2073.276]
  MoveL 893 to (3.42, 313.28, 130) mm, rotated rx -90 ry -25 rz -133.09 deg; joints [-2.628, -48.76, 103.313, 217.483, 108.441, -182.632, -2066.906]
  MoveL 894 to (10.42, 312.45, 120) mm, rotated rx -90 ry -25 rz -139.47 deg; joints [-2.992, -48.899, 103.589, 217.27, 108.422, -182.367, -2060.525]
  MoveL 895 to (17.25, 310.8, 110) mm, rotated rx -90 ry -25 rz -145.84 deg; joints [-3.358, -49.032, 103.86, 217.055, 108.404, -182.103, -2054.159]
  MoveL 896 to (23.78, 308.38, 100) mm, rotated rx -90 ry -25 rz -152.16 deg; joints [-3.725, -49.16, 104.124, 216.838, 108.386, -181.838, -2047.838]
  MoveL 897 to (29.89, 305.25, 90) mm, rotated rx -90 ry -25 rz -158.41 deg; joints [-4.093, -49.282, 104.382, 216.619, 108.369, -181.574, -2041.588]
  MoveL 898 to (35.48, 301.51, 80) mm, rotated rx -90 ry -25 rz -164.56 deg; joints [-4.463, -49.398, 104.635, 216.399, 108.352, -181.31, -2035.44]
  MoveL 899 to (40.49, 297.28, 70) mm, rotated rx -90 ry -25 rz -170.58 deg; joints [-4.834, -49.51, 104.881, 216.176, 108.336, -181.047, -2029.423]
  MoveL 900 to (44.86, 292.68, 60) mm, rotated rx -90 ry -25 rz -176.43 deg; joints [-5.207, -49.617, 105.121, 215.952, 108.319, -180.784, -2023.57]
  MoveL 901 to (48.58, 287.83, 50) mm, rotated rx -90 ry -25 rz 177.91 deg; joints [-5.581, -49.72, 105.355, 215.726, 108.302, -180.523, -2017.914]
  MoveL 902 to (51.63, 282.88, 40) mm, rotated rx -90 ry -25 rz 172.49 deg; joints [-5.956, -49.819, 105.582, 215.498, 108.283, -180.263, -2012.49]
  MoveL 903 to (54.06, 277.94, 30) mm, rotated rx -90 ry -25 rz 167.33 deg; joints [-6.332, -49.914, 105.804, 215.267, 108.263, -180.005, -2007.332]
  MoveL 904 to (55.91, 273.13, 20) mm, rotated rx -90 ry -25 rz 162.48 deg; joints [-6.709, -50.007, 106.019, 215.035, 108.241, -179.749, -2002.48]
  MoveL 905 to (57.23, 268.56, 10) mm, rotated rx -90 ry -25 rz 157.97 deg; joints [-7.088, -50.097, 106.227, 214.8, 108.218, -179.495, -1997.971]
  MoveL 906 to (58.12, 264.32, 0) mm, rotated rx -90 ry -25 rz 153.85 deg; joints [-7.468, -50.186, 106.43, 214.563, 108.191, -179.243, -1993.845]
  MoveL 907 to (-58.22, 263.67, 290) mm, rotated rx -90 ry -25 rz -53.21 deg; joints [2.992, -45.884, 98.039, 220.612, 108.694, -186.971, -2146.787]
  Set speed (60.0 mm/s)
  MoveL 908 to (-78.63, 259.66, 290) mm, rotated rx -90 ry -25 rz -47.01 deg; joints [2.992, -46.754, 97.943, 220.404, 107.959, -187.632, -2152.994]
  MoveL 909 to (58.12, 264.32, 0) mm, rotated rx -90 ry -25 rz 153.85 deg; joints [-7.468, -50.186, 106.43, 214.563, 108.191, -179.243, -1993.845]
  Set speed (60.0 mm/s)
  MoveL 910 to (76.17, 274.65, 0) mm, rotated rx -90 ry -25 rz 157.93 deg; joints [-7.468, -51.166, 106.328, 214.367, 107.299, -179.886, -1997.935]
  MoveL 911 to (58.12, 264.32, 0) mm, rotated rx -90 ry -25 rz 153.85 deg; joints [-7.468, -50.186, 106.43, 214.563, 108.191, -179.243, -1993.845]
  Set speed (60.0 mm/s)
  MoveL 912 to (57.23, 268.56, 10) mm, rotated rx -90 ry -25 rz 157.97 deg; joints [-7.088, -50.097, 106.227, 214.8, 108.218, -179.495, -1997.971]
  MoveL 913 to (55.91, 273.13, 20) mm, rotated rx -90 ry -25 rz 162.48 deg; joints [-6.709, -50.007, 106.019, 215.035, 108.241, -179.749, -2002.48]
  MoveL 914 to (54.06, 277.94, 30) mm, rotated rx -90 ry -25 rz 167.33 deg; joints [-6.332, -49.914, 105.804, 215.267, 108.263, -180.005, -2007.332]
  MoveL 915 to (51.63, 282.88, 40) mm, rotated rx -90 ry -25 rz 172.49 deg; joints [-5.956, -49.819, 105.582, 215.498, 108.283, -180.263, -2012.49]
  MoveL 916 to (48.58, 287.83, 50) mm, rotated rx -90 ry -25 rz 177.91 deg; joints [-5.581, -49.72, 105.355, 215.726, 108.302, -180.523, -2017.914]
  MoveL 917 to (44.86, 292.68, 60) mm, rotated rx -90 ry -25 rz -176.43 deg; joints [-5.207, -49.617, 105.121, 215.952, 108.319, -180.784, -2023.57]
  MoveL 918 to (40.49, 297.28, 70) mm, rotated rx -90 ry -25 rz -170.58 deg; joints [-4.834, -49.51, 104.881, 216.176, 108.336, -181.047, -2029.423]
  MoveL 919 to (35.48, 301.51, 80) mm, rotated rx -90 ry -25 rz -164.56 deg; joints [-4.463, -49.398, 104.635, 216.399, 108.352, -181.31, -2035.44]
  MoveL 920 to (29.89, 305.25, 90) mm, rotated rx -90 ry -25 rz -158.41 deg; joints [-4.093, -49.282, 104.382, 216.619, 108.369, -181.574, -2041.588]
  MoveL 921 to (23.78, 308.38, 100) mm, rotated rx -90 ry -25 rz -152.16 deg; joints [-3.725, -49.16, 104.124, 216.838, 108.386, -181.838, -2047.838]
  MoveL 922 to (17.25, 310.8, 110) mm, rotated rx -90 ry -25 rz -145.84 deg; joints [-3.358, -49.032, 103.86, 217.055, 108.404, -182.103, -2054.159]
  MoveL 923 to (10.42, 312.45, 120) mm, rotated rx -90 ry -25 rz -139.47 deg; joints [-2.992, -48.899, 103.589, 217.27, 108.422, -182.367, -2060.525]
  MoveL 924 to (3.42, 313.28, 130) mm, rotated rx -90 ry -25 rz -133.09 deg; joints [-2.628, -48.76, 103.313, 217.483, 108.441, -182.632, -2066.906]
  MoveL 925 to (-3.62, 313.27, 140) mm, rotated rx -90 ry -25 rz -126.72 deg; joints [-2.265, -48.614, 103.03, 217.695, 108.461, -182.896, -2073.276]
  MoveL 926 to (-10.57, 312.43, 150) mm, rotated rx -90 ry -25 rz -120.39 deg; joints [-1.904, -48.463, 102.742, 217.905, 108.481, -183.16, -2079.606]
  MoveL 927 to (-17.28, 310.79, 160) mm, rotated rx -90 ry -25 rz -114.13 deg; joints [-1.544, -48.306, 102.447, 218.113, 108.503, -183.424, -2085.87]
  MoveL 928 to (-23.65, 308.43, 170) mm, rotated rx -90 ry -25 rz -107.96 deg; joints [-1.185, -48.143, 102.146, 218.319, 108.524, -183.689, -2092.038]
  MoveL 929 to (-29.57, 305.43, 180) mm, rotated rx -90 ry -25 rz -101.92 deg; joints [-0.828, -47.975, 101.839, 218.524, 108.546, -183.953, -2098.081]
  MoveL 930 to (-34.96, 301.9, 190) mm, rotated rx -90 ry -25 rz -96.03 deg; joints [-0.473, -47.802, 101.526, 218.726, 108.567, -184.218, -2103.97]
  MoveL 931 to (-39.77, 297.95, 200) mm, rotated rx -90 ry -25 rz -90.33 deg; joints [-0.119, -47.624, 101.206, 218.926, 108.588, -184.485, -2109.672]
  MoveL 932 to (-43.95, 293.72, 210) mm, rotated rx -90 ry -25 rz -84.84 deg; joints [0.233, -47.443, 100.881, 219.124, 108.608, -184.752, -2115.156]
  MoveL 933 to (-47.51, 289.33, 220) mm, rotated rx -90 ry -25 rz -79.61 deg; joints [0.584, -47.257, 100.549, 219.32, 108.627, -185.021, -2120.386]
  MoveL 934 to (-50.46, 284.91, 230) mm, rotated rx -90 ry -25 rz -74.67 deg; joints [0.933, -47.068, 100.21, 219.513, 108.644, -185.292, -2125.328]
  MoveL 935 to (-52.84, 280.57, 240) mm, rotated rx -90 ry -25 rz -70.06 deg; joints [1.28, -46.876, 99.865, 219.703, 108.659, -185.564, -2129.944]
  MoveL 936 to (-54.69, 276.44, 250) mm, rotated rx -90 ry -25 rz -65.8 deg; joints [1.626, -46.682, 99.513, 219.891, 108.672, -185.84, -2134.197]
  MoveL 937 to (-56.08, 272.6, 260) mm, rotated rx -90 ry -25 rz -61.95 deg; joints [1.97, -46.485, 99.155, 220.076, 108.682, -186.118, -2138.047]
  MoveL 938 to (-57.08, 269.15, 270) mm, rotated rx -90 ry -25 rz -58.54 deg; joints [2.312, -46.286, 98.79, 220.257, 108.689, -186.399, -2141.455]
  MoveL 939 to (-57.77, 266.15, 280) mm, rotated rx -90 ry -25 rz -55.62 deg; joints [2.653, -46.086, 98.418, 220.436, 108.693, -186.683, -2144.382]
  MoveL 940 to (-58.22, 263.67, 290) mm, rotated rx -90 ry -25 rz -53.21 deg; joints [2.992, -45.884, 98.039, 220.612, 108.694, -186.971, -2146.787]
  MoveL 941 to (-78.63, 259.66, 290) mm, rotated rx -90 ry -25 rz -47.01 deg; joints [2.992, -46.754, 97.943, 220.404, 107.959, -187.632, -2152.994]
  Set speed (60.0 mm/s)
  MoveL 942 to (-78.34, 263.02, 280) mm, rotated rx -90 ry -25 rz -49.44 deg; joints [2.653, -46.959, 98.321, 220.229, 107.954, -187.345, -2150.563]
  MoveL 943 to (-77.78, 267.1, 270) mm, rotated rx -90 ry -25 rz -52.4 deg; joints [2.312, -47.163, 98.693, 220.05, 107.945, -187.06, -2147.603]
  MoveL 944 to (-76.86, 271.82, 260) mm, rotated rx -90 ry -25 rz -55.85 deg; joints [1.97, -47.365, 99.057, 219.868, 107.933, -186.779, -2144.153]
  MoveL 945 to (-75.48, 277.1, 250) mm, rotated rx -90 ry -25 rz -59.75 deg; joints [1.626, -47.564, 99.415, 219.683, 107.918, -186.501, -2140.252]
  MoveL 946 to (-73.51, 282.82, 240) mm, rotated rx -90 ry -25 rz -64.06 deg; joints [1.28, -47.762, 99.766, 219.496, 107.901, -186.225, -2135.94]
  MoveL 947 to (-70.88, 288.88, 230) mm, rotated rx -90 ry -25 rz -68.74 deg; joints [0.933, -47.957, 100.111, 219.305, 107.88, -185.952, -2131.255]
  MoveL 948 to (-67.49, 295.12, 220) mm, rotated rx -90 ry -25 rz -73.76 deg; joints [0.584, -48.15, 100.449, 219.113, 107.858, -185.682, -2126.236]
  MoveL 949 to (-63.28, 301.4, 210) mm, rotated rx -90 ry -25 rz -79.08 deg; joints [0.233, -48.339, 100.78, 218.917, 107.834, -185.413, -2120.918]
  MoveL 950 to (-58.22, 307.54, 200) mm, rotated rx -90 ry -25 rz -84.66 deg; joints [-0.119, -48.525, 101.105, 218.72, 107.808, -185.146, -2115.34]
  MoveL 951 to (-52.31, 313.38, 190) mm, rotated rx -90 ry -25 rz -90.47 deg; joints [-0.473, -48.707, 101.424, 218.52, 107.781, -184.88, -2109.535]
  MoveL 952 to (-45.56, 318.73, 180) mm, rotated rx -90 ry -25 rz -96.46 deg; joints [-0.828, -48.884, 101.737, 218.318, 107.754, -184.615, -2103.538]
  MoveL 953 to (-38.04, 323.45, 170) mm, rotated rx -90 ry -25 rz -102.62 deg; joints [-1.185, -49.056, 102.043, 218.113, 107.726, -184.35, -2097.381]
  MoveL 954 to (-29.85, 327.37, 160) mm, rotated rx -90 ry -25 rz -108.9 deg; joints [-1.544, -49.223, 102.343, 217.907, 107.698, -184.086, -2091.097]
  MoveL 955 to (-21.11, 330.36, 150) mm, rotated rx -90 ry -25 rz -115.28 deg; joints [-1.904, -49.385, 102.637, 217.7, 107.67, -183.822, -2084.715]
  MoveL 956 to (-11.96, 332.32, 140) mm, rotated rx -90 ry -25 rz -121.73 deg; joints [-2.265, -49.541, 102.926, 217.49, 107.643, -183.558, -2078.268]
  MoveL 957 to (-2.59, 333.2, 130) mm, rotated rx -90 ry -25 rz -128.22 deg; joints [-2.628, -49.691, 103.208, 217.278, 107.617, -183.293, -2071.782]
  MoveL 958 to (6.83, 332.94, 120) mm, rotated rx -90 ry -25 rz -134.71 deg; joints [-2.992, -49.835, 103.484, 217.065, 107.592, -183.029, -2065.289]
  MoveL 959 to (16.13, 331.57, 110) mm, rotated rx -90 ry -25 rz -141.18 deg; joints [-3.358, -49.973, 103.754, 216.851, 107.568, -182.764, -2058.817]
  MoveL 960 to (25.11, 329.13, 100) mm, rotated rx -90 ry -25 rz -147.6 deg; joints [-3.725, -50.105, 104.019, 216.634, 107.544, -182.499, -2052.396]
  MoveL 961 to (33.62, 325.71, 90) mm, rotated rx -90 ry -25 rz -153.95 deg; joints [-4.093, -50.231, 104.277, 216.416, 107.521, -182.234, -2046.054]
  MoveL 962 to (41.52, 321.41, 80) mm, rotated rx -90 ry -25 rz -160.18 deg; joints [-4.463, -50.352, 104.53, 216.196, 107.499, -181.969, -2039.824]
  MoveL 963 to (48.7, 316.39, 70) mm, rotated rx -90 ry -25 rz -166.26 deg; joints [-4.834, -50.468, 104.776, 215.974, 107.477, -181.704, -2033.735]
  MoveL 964 to (55.08, 310.79, 60) mm, rotated rx -90 ry -25 rz -172.18 deg; joints [-5.207, -50.578, 105.016, 215.751, 107.455, -181.44, -2027.821]
  MoveL 965 to (60.61, 304.79, 50) mm, rotated rx -90 ry -25 rz -177.89 deg; joints [-5.581, -50.685, 105.251, 215.525, 107.432, -181.177, -2022.113]
  MoveL 966 to (65.29, 298.57, 40) mm, rotated rx -90 ry -25 rz 176.65 deg; joints [-5.956, -50.787, 105.479, 215.298, 107.409, -180.915, -2016.648]
  MoveL 967 to (69.12, 292.29, 30) mm, rotated rx -90 ry -25 rz 171.46 deg; joints [-6.332, -50.886, 105.701, 215.068, 107.384, -180.655, -2011.461]
  MoveL 968 to (72.16, 286.11, 20) mm, rotated rx -90 ry -25 rz 166.59 deg; joints [-6.709, -50.982, 105.916, 214.837, 107.358, -180.397, -2006.587]
  MoveL 969 to (74.48, 280.19, 10) mm, rotated rx -90 ry -25 rz 162.07 deg; joints [-7.088, -51.075, 106.125, 214.603, 107.33, -180.14, -2002.066]
  MoveL 970 to (76.17, 274.65, 0) mm, rotated rx -90 ry -25 rz 157.93 deg; joints [-7.468, -51.166, 106.328, 214.367, 107.299, -179.886, -1997.935]
  MoveL 971 to (-78.63, 259.66, 290) mm, rotated rx -90 ry -25 rz -47.01 deg; joints [2.992, -46.754, 97.943, 220.404, 107.959, -187.632, -2152.994]
  Set speed (60.0 mm/s)
  MoveL 972 to (-58.93, 252.99, 290) mm, rotated rx -90 ry -25 rz -42.9 deg; joints [2.992, -45.848, 98.043, 220.621, 108.724, -186.944, -2157.096]
  MoveL 973 to (76.17, 274.65, 0) mm, rotated rx -90 ry -25 rz 157.93 deg; joints [-7.468, -51.166, 106.328, 214.367, 107.299, -179.886, -1997.935]
  Set speed (60.0 mm/s)
  MoveL 974 to (55.37, 274.67, 0) mm, rotated rx -90 ry -25 rz 164.01 deg; joints [-7.468, -50.223, 106.427, 214.556, 108.158, -179.268, -2004.014]
  MoveL 975 to (76.17, 274.65, 0) mm, rotated rx -90 ry -25 rz 157.93 deg; joints [-7.468, -51.166, 106.328, 214.367, 107.299, -179.886, -1997.935]
  Set speed (60.0 mm/s)
  MoveL 976 to (74.48, 280.19, 10) mm, rotated rx -90 ry -25 rz 162.07 deg; joints [-7.088, -51.075, 106.125, 214.603, 107.33, -180.14, -2002.066]
  MoveL 977 to (72.16, 286.11, 20) mm, rotated rx -90 ry -25 rz 166.59 deg; joints [-6.709, -50.982, 105.916, 214.837, 107.358, -180.397, -2006.587]
  MoveL 978 to (69.12, 292.29, 30) mm, rotated rx -90 ry -25 rz 171.46 deg; joints [-6.332, -50.886, 105.701, 215.068, 107.384, -180.655, -2011.461]
  MoveL 979 to (65.29, 298.57, 40) mm, rotated rx -90 ry -25 rz 176.65 deg; joints [-5.956, -50.787, 105.479, 215.298, 107.409, -180.915, -2016.648]
  MoveL 980 to (60.61, 304.79, 50) mm, rotated rx -90 ry -25 rz -177.89 deg; joints [-5.581, -50.685, 105.251, 215.525, 107.432, -181.177, -2022.113]
  MoveL 981 to (55.08, 310.79, 60) mm, rotated rx -90 ry -25 rz -172.18 deg; joints [-5.207, -50.578, 105.016, 215.751, 107.455, -181.44, -2027.821]
  MoveL 982 to (48.7, 316.39, 70) mm, rotated rx -90 ry -25 rz -166.26 deg; joints [-4.834, -50.468, 104.776, 215.974, 107.477, -181.704, -2033.735]
  MoveL 983 to (41.52, 321.41, 80) mm, rotated rx -90 ry -25 rz -160.18 deg; joints [-4.463, -50.352, 104.53, 216.196, 107.499, -181.969, -2039.824]
  MoveL 984 to (33.62, 325.71, 90) mm, rotated rx -90 ry -25 rz -153.95 deg; joints [-4.093, -50.231, 104.277, 216.416, 107.521, -182.234, -2046.054]
  MoveL 985 to (25.11, 329.13, 100) mm, rotated rx -90 ry -25 rz -147.6 deg; joints [-3.725, -50.105, 104.019, 216.634, 107.544, -182.499, -2052.396]
  MoveL 986 to (16.13, 331.57, 110) mm, rotated rx -90 ry -25 rz -141.18 deg; joints [-3.358, -49.973, 103.754, 216.851, 107.568, -182.764, -2058.817]
  MoveL 987 to (6.83, 332.94, 120) mm, rotated rx -90 ry -25 rz -134.71 deg; joints [-2.992, -49.835, 103.484, 217.065, 107.592, -183.029, -2065.289]
  MoveL 988 to (-2.59, 333.2, 130) mm, rotated rx -90 ry -25 rz -128.22 deg; joints [-2.628, -49.691, 103.208, 217.278, 107.617, -183.293, -2071.782]
  MoveL 989 to (-11.96, 332.32, 140) mm, rotated rx -90 ry -25 rz -121.73 deg; joints [-2.265, -49.541, 102.926, 217.49, 107.643, -183.558, -2078.268]
  MoveL 990 to (-21.11, 330.36, 150) mm, rotated rx -90 ry -25 rz -115.28 deg; joints [-1.904, -49.385, 102.637, 217.7, 107.67, -183.822, -2084.715]
  MoveL 991 to (-29.85, 327.37, 160) mm, rotated rx -90 ry -25 rz -108.9 deg; joints [-1.544, -49.223, 102.343, 217.907, 107.698, -184.086, -2091.097]
  MoveL 992 to (-38.04, 323.45, 170) mm, rotated rx -90 ry -25 rz -102.62 deg; joints [-1.185, -49.056, 102.043, 218.113, 107.726, -184.35, -2097.381]
  MoveL 993 to (-45.56, 318.73, 180) mm, rotated rx -90 ry -25 rz -96.46 deg; joints [-0.828, -48.884, 101.737, 218.318, 107.754, -184.615, -2103.538]
  MoveL 994 to (-52.31, 313.38, 190) mm, rotated rx -90 ry -25 rz -90.47 deg; joints [-0.473, -48.707, 101.424, 218.52, 107.781, -184.88, -2109.535]
  MoveL 995 to (-58.22, 307.54, 200) mm, rotated rx -90 ry -25 rz -84.66 deg; joints [-0.119, -48.525, 101.105, 218.72, 107.808, -185.146, -2115.34]
  MoveL 996 to (-63.28, 301.4, 210) mm, rotated rx -90 ry -25 rz -79.08 deg; joints [0.233, -48.339, 100.78, 218.917, 107.834, -185.413, -2120.918]
  MoveL 997 to (-67.49, 295.12, 220) mm, rotated rx -90 ry -25 rz -73.76 deg; joints [0.584, -48.15, 100.449, 219.113, 107.858, -185.682, -2126.236]
  MoveL 998 to (-70.88, 288.88, 230) mm, rotated rx -90 ry -25 rz -68.74 deg; joints [0.933, -47.957, 100.111, 219.305, 107.88, -185.952, -2131.255]
  MoveL 999 to (-73.51, 282.82, 240) mm, rotated rx -90 ry -25 rz -64.06 deg; joints [1.28, -47.762, 99.766, 219.496, 107.901, -186.225, -2135.94]
  MoveL 1000 to (-75.48, 277.1, 250) mm, rotated rx -90 ry -25 rz -59.75 deg; joints [1.626, -47.564, 99.415, 219.683, 107.918, -186.501, -2140.252]
  MoveL 1001 to (-76.86, 271.82, 260) mm, rotated rx -90 ry -25 rz -55.85 deg; joints [1.97, -47.365, 99.057, 219.868, 107.933, -186.779, -2144.153]
  MoveL 1002 to (-77.78, 267.1, 270) mm, rotated rx -90 ry -25 rz -52.4 deg; joints [2.312, -47.163, 98.693, 220.05, 107.945, -187.06, -2147.603]
  MoveL 1003 to (-78.34, 263.02, 280) mm, rotated rx -90 ry -25 rz -49.44 deg; joints [2.653, -46.959, 98.321, 220.229, 107.954, -187.345, -2150.563]
  MoveL 1004 to (-78.63, 259.66, 290) mm, rotated rx -90 ry -25 rz -47.01 deg; joints [2.992, -46.754, 97.943, 220.404, 107.959, -187.632, -2152.994]
  MoveL 1005 to (-58.93, 252.99, 290) mm, rotated rx -90 ry -25 rz -42.9 deg; joints [2.992, -45.848, 98.043, 220.621, 108.724, -186.944, -2157.096]
  Set speed (60.0 mm/s)
  MoveL 1006 to (-58.94, 255.51, 280) mm, rotated rx -90 ry -25 rz -45.34 deg; joints [2.653, -46.05, 98.421, 220.445, 108.723, -186.656, -2154.659]
  MoveL 1007 to (-58.8, 258.59, 270) mm, rotated rx -90 ry -25 rz -48.31 deg; joints [2.312, -46.251, 98.793, 220.266, 108.719, -186.372, -2151.694]
  MoveL 1008 to (-58.44, 262.16, 260) mm, rotated rx -90 ry -25 rz -51.76 deg; joints [1.97, -46.45, 99.158, 220.084, 108.711, -186.092, -2148.242]
  MoveL 1009 to (-57.77, 266.19, 250) mm, rotated rx -90 ry -25 rz -55.66 deg; joints [1.626, -46.647, 99.516, 219.899, 108.701, -185.814, -2144.344]
  MoveL 1010 to (-56.69, 270.59, 240) mm, rotated rx -90 ry -25 rz -59.96 deg; joints [1.28, -46.843, 99.868, 219.711, 108.687, -185.54, -2140.04]
  MoveL 1011 to (-55.14, 275.28, 230) mm, rotated rx -90 ry -25 rz -64.63 deg; joints [0.933, -47.036, 100.213, 219.52, 108.671, -185.268, -2135.371]
  MoveL 1012 to (-53.04, 280.16, 220) mm, rotated rx -90 ry -25 rz -69.62 deg; joints [0.584, -47.227, 100.551, 219.327, 108.653, -184.998, -2130.377]
  MoveL 1013 to (-50.33, 285.12, 210) mm, rotated rx -90 ry -25 rz -74.91 deg; joints [0.233, -47.414, 100.883, 219.131, 108.633, -184.731, -2125.094]
  MoveL 1014 to (-46.98, 290.04, 200) mm, rotated rx -90 ry -25 rz -80.44 deg; joints [-0.119, -47.598, 101.209, 218.932, 108.611, -184.466, -2119.561]
  MoveL 1015 to (-42.97, 294.79, 190) mm, rotated rx -90 ry -25 rz -86.19 deg; joints [-0.473, -47.778, 101.528, 218.731, 108.588, -184.201, -2113.811]
  MoveL 1016 to (-38.31, 299.24, 180) mm, rotated rx -90 ry -25 rz -92.12 deg; joints [-0.828, -47.955, 101.841, 218.528, 108.564, -183.938, -2107.881]
  MoveL 1017 to (-33.03, 303.26, 170) mm, rotated rx -90 ry -25 rz -98.2 deg; joints [-1.185, -48.126, 102.148, 218.323, 108.539, -183.676, -2101.801]
  MoveL 1018 to (-27.19, 306.74, 160) mm, rotated rx -90 ry -25 rz -104.4 deg; joints [-1.544, -48.292, 102.448, 218.116, 108.514, -183.415, -2095.603]
  MoveL 1019 to (-20.88, 309.56, 150) mm, rotated rx -90 ry -25 rz -110.68 deg; joints [-1.904, -48.453, 102.742, 217.907, 108.49, -183.153, -2089.318]
  MoveL 1020 to (-14.2, 311.65, 140) mm, rotated rx -90 ry -25 rz -117.03 deg; joints [-2.265, -48.609, 103.031, 217.696, 108.465, -182.892, -2082.972]
  MoveL 1021 to (-7.28, 312.93, 130) mm, rotated rx -90 ry -25 rz -123.4 deg; joints [-2.628, -48.758, 103.313, 217.483, 108.442, -182.631, -2076.596]
  MoveL 1022 to (-0.24, 313.38, 120) mm, rotated rx -90 ry -25 rz -129.78 deg; joints [-2.992, -48.902, 103.589, 217.269, 108.419, -182.369, -2070.217]
  MoveL 1023 to (6.77, 312.99, 110) mm, rotated rx -90 ry -25 rz -136.14 deg; joints [-3.358, -49.04, 103.859, 217.053, 108.397, -182.108, -2063.862]
  MoveL 1024 to (13.63, 311.79, 100) mm, rotated rx -90 ry -25 rz -142.44 deg; joints [-3.725, -49.171, 104.123, 216.835, 108.376, -181.846, -2057.558]
  MoveL 1025 to (20.21, 309.81, 90) mm, rotated rx -90 ry -25 rz -148.67 deg; joints [-4.093, -49.297, 104.381, 216.616, 108.356, -181.584, -2051.334]
  MoveL 1026 to (26.38, 307.15, 80) mm, rotated rx -90 ry -25 rz -154.78 deg; joints [-4.463, -49.418, 104.633, 216.395, 108.336, -181.323, -2045.218]
  MoveL 1027 to (32.08, 303.89, 70) mm, rotated rx -90 ry -25 rz -160.76 deg; joints [-4.834, -49.533, 104.879, 216.172, 108.316, -181.062, -2039.241]
  MoveL 1028 to (37.21, 300.16, 60) mm, rotated rx -90 ry -25 rz -166.57 deg; joints [-5.207, -49.643, 105.118, 215.947, 108.296, -180.801, -2033.432]
  MoveL 1029 to (41.73, 296.07, 50) mm, rotated rx -90 ry -25 rz -172.18 deg; joints [-5.581, -49.748, 105.352, 215.72, 108.276, -180.542, -2027.825]
  MoveL 1030 to (45.64, 291.75, 40) mm, rotated rx -90 ry -25 rz -177.55 deg; joints [-5.956, -49.85, 105.579, 215.491, 108.256, -180.284, -2022.451]
  MoveL 1031 to (48.92, 287.33, 30) mm, rotated rx -90 ry -25 rz 177.35 deg; joints [-6.332, -49.947, 105.801, 215.26, 108.234, -180.027, -2017.347]
  MoveL 1032 to (51.6, 282.93, 20) mm, rotated rx -90 ry -25 rz 172.55 deg; joints [-6.709, -50.042, 106.016, 215.028, 108.21, -179.772, -2012.547]
  MoveL 1033 to (53.73, 278.68, 10) mm, rotated rx -90 ry -25 rz 168.09 deg; joints [-7.088, -50.134, 106.224, 214.793, 108.185, -179.518, -2008.09]
  MoveL 1034 to (55.37, 274.67, 0) mm, rotated rx -90 ry -25 rz 164.01 deg; joints [-7.468, -50.223, 106.427, 214.556, 108.158, -179.268, -2004.014]
  MoveL 1035 to (-58.93, 252.99, 290) mm, rotated rx -90 ry -25 rz -42.9 deg; joints [2.992, -45.848, 98.043, 220.621, 108.724, -186.944, -2157.096]
  Set speed (60.0 mm/s)
  MoveL 1036 to (-37.11, 208.63, 290) mm, rotated rx -90 ry -25 rz 8.11 deg; joints [2.992, -45.692, 98.056, 220.659, 108.852, -186.827, -2208.107]
  MoveL 1037 to (55.37, 274.67, 0) mm, rotated rx -90 ry -25 rz 164.01 deg; joints [-7.468, -50.223, 106.427, 214.556, 108.158, -179.268, -2364.014]
  Set speed (60.0 mm/s)
  MoveL 1038 to (20.49, 309.71, 0) mm, rotated rx -90 ry -25 rz -148.94 deg; joints [-7.468, -50.346, 106.416, 214.531, 108.048, -179.347, -2411.057]
  MoveL 1039 to (55.37, 274.67, 0) mm, rotated rx -90 ry -25 rz 164.01 deg; joints [-7.468, -50.223, 106.427, 214.556, 108.158, -179.268, -2364.014]
  Set speed (60.0 mm/s)
  MoveL 1040 to (53.73, 278.68, 10) mm, rotated rx -90 ry -25 rz 168.09 deg; joints [-7.088, -50.134, 106.224, 214.793, 108.185, -179.518, -2368.09]
  MoveL 1041 to (51.6, 282.93, 20) mm, rotated rx -90 ry -25 rz 172.55 deg; joints [-6.709, -50.042, 106.016, 215.028, 108.21, -179.772, -2372.547]
  MoveL 1042 to (48.92, 287.33, 30) mm, rotated rx -90 ry -25 rz 177.35 deg; joints [-6.332, -49.947, 105.801, 215.26, 108.234, -180.027, -2377.347]
  MoveL 1043 to (45.64, 291.75, 40) mm, rotated rx -90 ry -25 rz -177.55 deg; joints [-5.956, -49.85, 105.579, 215.491, 108.256, -180.284, -2382.451]
  MoveL 1044 to (41.73, 296.07, 50) mm, rotated rx -90 ry -25 rz -172.18 deg; joints [-5.581, -49.748, 105.352, 215.72, 108.276, -180.542, -2387.825]
  MoveL 1045 to (37.21, 300.16, 60) mm, rotated rx -90 ry -25 rz -166.57 deg; joints [-5.207, -49.643, 105.118, 215.947, 108.296, -180.801, -2393.432]
  MoveL 1046 to (32.08, 303.89, 70) mm, rotated rx -90 ry -25 rz -160.76 deg; joints [-4.834, -49.533, 104.879, 216.172, 108.316, -181.062, -2399.241]
  MoveL 1047 to (26.38, 307.15, 80) mm, rotated rx -90 ry -25 rz -154.78 deg; joints [-4.463, -49.418, 104.633, 216.395, 108.336, -181.323, -2405.218]
  MoveL 1048 to (20.21, 309.81, 90) mm, rotated rx -90 ry -25 rz -148.67 deg; joints [-4.093, -49.297, 104.381, 216.616, 108.356, -181.584, -2411.334]
  MoveL 1049 to (13.63, 311.79, 100) mm, rotated rx -90 ry -25 rz -142.44 deg; joints [-3.725, -49.171, 104.123, 216.835, 108.376, -181.846, -2417.558]
  MoveL 1050 to (6.77, 312.99, 110) mm, rotated rx -90 ry -25 rz -136.14 deg; joints [-3.358, -49.04, 103.859, 217.053, 108.397, -182.108, -2423.862]
  MoveL 1051 to (-0.24, 313.38, 120) mm, rotated rx -90 ry -25 rz -129.78 deg; joints [-2.992, -48.902, 103.589, 217.269, 108.419, -182.369, -2430.217]
  MoveL 1052 to (-7.28, 312.93, 130) mm, rotated rx -90 ry -25 rz -123.4 deg; joints [-2.628, -48.758, 103.313, 217.483, 108.442, -182.631, -2436.596]
  MoveL 1053 to (-14.2, 311.65, 140) mm, rotated rx -90 ry -25 rz -117.03 deg; joints [-2.265, -48.609, 103.031, 217.696, 108.465, -182.892, -2442.972]
  MoveL 1054 to (-20.88, 309.56, 150) mm, rotated rx -90 ry -25 rz -110.68 deg; joints [-1.904, -48.453, 102.742, 217.907, 108.49, -183.153, -2449.318]
  MoveL 1055 to (-27.19, 306.74, 160) mm, rotated rx -90 ry -25 rz -104.4 deg; joints [-1.544, -48.292, 102.448, 218.116, 108.514, -183.415, -2455.603]
  MoveL 1056 to (-33.03, 303.26, 170) mm, rotated rx -90 ry -25 rz -98.2 deg; joints [-1.185, -48.126, 102.148, 218.323, 108.539, -183.676, -2461.801]
  MoveL 1057 to (-38.31, 299.24, 180) mm, rotated rx -90 ry -25 rz -92.12 deg; joints [-0.828, -47.955, 101.841, 218.528, 108.564, -183.938, -2467.881]
  MoveL 1058 to (-42.97, 294.79, 190) mm, rotated rx -90 ry -25 rz -86.19 deg; joints [-0.473, -47.778, 101.528, 218.731, 108.588, -184.201, -2473.811]
  MoveL 1059 to (-46.98, 290.04, 200) mm, rotated rx -90 ry -25 rz -80.44 deg; joints [-0.119, -47.598, 101.209, 218.932, 108.611, -184.466, -2479.561]
  MoveL 1060 to (-50.33, 285.12, 210) mm, rotated rx -90 ry -25 rz -74.91 deg; joints [0.233, -47.414, 100.883, 219.131, 108.633, -184.731, -2485.094]
  MoveL 1061 to (-53.04, 280.16, 220) mm, rotated rx -90 ry -25 rz -69.62 deg; joints [0.584, -47.227, 100.551, 219.327, 108.653, -184.998, -2490.377]
  MoveL 1062 to (-55.14, 275.28, 230) mm, rotated rx -90 ry -25 rz -64.63 deg; joints [0.933, -47.036, 100.213, 219.52, 108.671, -185.268, -2495.371]
  MoveL 1063 to (-56.69, 270.59, 240) mm, rotated rx -90 ry -25 rz -59.96 deg; joints [1.28, -46.843, 99.868, 219.711, 108.687, -185.54, -2500.04]
  MoveL 1064 to (-57.77, 266.19, 250) mm, rotated rx -90 ry -25 rz -55.66 deg; joints [1.626, -46.647, 99.516, 219.899, 108.701, -185.814, -2504.344]
  MoveL 1065 to (-58.44, 262.16, 260) mm, rotated rx -90 ry -25 rz -51.76 deg; joints [1.97, -46.45, 99.158, 220.084, 108.711, -186.092, -2508.242]
  MoveL 1066 to (-58.8, 258.59, 270) mm, rotated rx -90 ry -25 rz -48.31 deg; joints [2.312, -46.251, 98.793, 220.266, 108.719, -186.372, -2511.694]
  MoveL 1067 to (-58.94, 255.51, 280) mm, rotated rx -90 ry -25 rz -45.34 deg; joints [2.653, -46.05, 98.421, 220.445, 108.723, -186.656, -2514.659]
  MoveL 1068 to (-58.93, 252.99, 290) mm, rotated rx -90 ry -25 rz -42.9 deg; joints [2.992, -45.848, 98.043, 220.621, 108.724, -186.944, -2517.096]
  MoveL 1069 to (-37.11, 208.63, 290) mm, rotated rx -90 ry -25 rz 8.11 deg; joints [2.992, -45.692, 98.056, 220.659, 108.852, -186.827, -2568.107]
  Set speed (60.0 mm/s)
  MoveL 1070 to (-39.03, 210.26, 280) mm, rotated rx -90 ry -25 rz 5.51 deg; joints [2.653, -45.891, 98.435, 220.483, 108.854, -186.538, -2565.515]
  MoveL 1071 to (-41.29, 212.35, 270) mm, rotated rx -90 ry -25 rz 2.36 deg; joints [2.312, -46.089, 98.807, 220.305, 108.853, -186.252, -2562.358]
  MoveL 1072 to (-43.78, 214.95, 260) mm, rotated rx -90 ry -25 rz -1.32 deg; joints [1.97, -46.284, 99.173, 220.123, 108.849, -185.969, -2558.681]
  MoveL 1073 to (-46.4, 218.08, 250) mm, rotated rx -90 ry -25 rz -5.47 deg; joints [1.626, -46.479, 99.531, 219.939, 108.841, -185.69, -2554.527]
  MoveL 1074 to (-49.06, 221.75, 240) mm, rotated rx -90 ry -25 rz -10.06 deg; joints [1.28, -46.672, 99.883, 219.751, 108.83, -185.414, -2549.94]
  MoveL 1075 to (-51.62, 225.97, 230) mm, rotated rx -90 ry -25 rz -15.04 deg; joints [0.933, -46.864, 100.228, 219.56, 108.815, -185.142, -2544.964]
  MoveL 1076 to (-53.98, 230.73, 220) mm, rotated rx -90 ry -25 rz -20.35 deg; joints [0.584, -47.055, 100.567, 219.367, 108.797, -184.873, -2539.646]
  MoveL 1077 to (-56, 236.01, 210) mm, rotated rx -90 ry -25 rz -25.97 deg; joints [0.233, -47.244, 100.899, 219.17, 108.776, -184.608, -2534.028]
  MoveL 1078 to (-57.57, 241.75, 200) mm, rotated rx -90 ry -25 rz -31.84 deg; joints [-0.119, -47.432, 101.224, 218.971, 108.752, -184.345, -2528.155]
  MoveL 1079 to (-58.59, 247.88, 190) mm, rotated rx -90 ry -25 rz -37.93 deg; joints [-0.473, -47.618, 101.543, 218.768, 108.724, -184.086, -2522.068]
  MoveL 1080 to (-58.95, 254.32, 180) mm, rotated rx -90 ry -25 rz -44.19 deg; joints [-0.828, -47.801, 101.855, 218.563, 108.694, -183.828, -2515.809]
  MoveL 1081 to (-58.59, 260.95, 170) mm, rotated rx -90 ry -25 rz -50.58 deg; joints [-1.185, -47.982, 102.161, 218.356, 108.662, -183.573, -2509.416]
  MoveL 1082 to (-57.45, 267.65, 160) mm, rotated rx -90 ry -25 rz -57.07 deg; joints [-1.544, -48.16, 102.46, 218.146, 108.628, -183.32, -2502.926]
  MoveL 1083 to (-55.51, 274.28, 150) mm, rotated rx -90 ry -25 rz -63.63 deg; joints [-1.904, -48.334, 102.753, 217.934, 108.592, -183.069, -2496.375]
  MoveL 1084 to (-52.77, 280.72, 140) mm, rotated rx -90 ry -25 rz -70.2 deg; joints [-2.265, -48.505, 103.04, 217.719, 108.556, -182.819, -2489.796]
  MoveL 1085 to (-49.26, 286.82, 130) mm, rotated rx -90 ry -25 rz -76.78 deg; joints [-2.628, -48.671, 103.321, 217.503, 108.518, -182.569, -2483.221]
  MoveL 1086 to (-45.04, 292.47, 120) mm, rotated rx -90 ry -25 rz -83.32 deg; joints [-2.992, -48.832, 103.595, 217.285, 108.48, -182.32, -2476.68]
  MoveL 1087 to (-40.19, 297.56, 110) mm, rotated rx -90 ry -25 rz -89.8 deg; joints [-3.358, -48.988, 103.864, 217.064, 108.442, -182.072, -2470.201]
  MoveL 1088 to (-34.83, 302, 100) mm, rotated rx -90 ry -25 rz -96.19 deg; joints [-3.725, -49.138, 104.126, 216.842, 108.405, -181.823, -2463.814]
  MoveL 1089 to (-29.06, 305.72, 90) mm, rotated rx -90 ry -25 rz -102.46 deg; joints [-4.093, -49.283, 104.382, 216.619, 108.368, -181.575, -2457.545]
  MoveL 1090 to (-23.03, 308.7, 80) mm, rotated rx -90 ry -25 rz -108.58 deg; joints [-4.463, -49.423, 104.632, 216.393, 108.331, -181.327, -2451.421]
  MoveL 1091 to (-16.86, 310.92, 70) mm, rotated rx -90 ry -25 rz -114.53 deg; joints [-4.834, -49.556, 104.876, 216.166, 108.295, -181.078, -2445.47]
  MoveL 1092 to (-10.69, 312.41, 60) mm, rotated rx -90 ry -25 rz -120.28 deg; joints [-5.207, -49.684, 105.115, 215.938, 108.259, -180.83, -2439.72]
  MoveL 1093 to (-4.64, 313.2, 50) mm, rotated rx -90 ry -25 rz -125.8 deg; joints [-5.581, -49.807, 105.347, 215.708, 108.224, -180.581, -2434.198]
  MoveL 1094 to (1.18, 313.37, 40) mm, rotated rx -90 ry -25 rz -131.07 deg; joints [-5.956, -49.924, 105.573, 215.476, 108.19, -180.333, -2428.933]
  MoveL 1095 to (6.67, 313.01, 30) mm, rotated rx -90 ry -25 rz -136.04 deg; joints [-6.332, -50.036, 105.793, 215.242, 108.155, -180.085, -2423.955]
  MoveL 1096 to (11.76, 312.2, 20) mm, rotated rx -90 ry -25 rz -140.7 deg; joints [-6.709, -50.143, 106.006, 215.007, 108.12, -179.838, -2419.296]
  MoveL 1097 to (16.38, 311.06, 10) mm, rotated rx -90 ry -25 rz -145.01 deg; joints [-7.088, -50.246, 106.214, 214.77, 108.084, -179.592, -2414.985]
  MoveL 1098 to (20.49, 309.71, 0) mm, rotated rx -90 ry -25 rz -148.94 deg; joints [-7.468, -50.346, 106.416, 214.531, 108.048, -179.347, -2411.057]
  MoveL 1099 to (-37.11, 208.63, 290) mm, rotated rx -90 ry -25 rz 8.11 deg; joints [2.992, -45.692, 98.056, 220.659, 108.852, -186.827, -2568.107]
  Set speed (60.0 mm/s)
  MoveL 1100 to (-43.85, 188.95, 290) mm, rotated rx -90 ry -25 rz 14.31 deg; joints [2.992, -46.574, 97.966, 220.447, 108.114, -187.494, -2574.314]
  MoveL 1101 to (20.49, 309.71, 0) mm, rotated rx -90 ry -25 rz -148.94 deg; joints [-7.468, -50.346, 106.416, 214.531, 108.048, -179.347, -2411.057]
  Set speed (60.0 mm/s)
  MoveL 1102 to (20.57, 330.51, 0) mm, rotated rx -90 ry -25 rz -144.34 deg; joints [-7.468, -51.311, 106.31, 214.338, 107.164, -179.983, -2415.665]
  MoveL 1103 to (20.49, 309.71, 0) mm, rotated rx -90 ry -25 rz -148.94 deg; joints [-7.468, -50.346, 106.416, 214.531, 108.048, -179.347, -2411.057]
  Set speed (60.0 mm/s)
  MoveL 1104 to (16.38, 311.06, 10) mm, rotated rx -90 ry -25 rz -145.01 deg; joints [-7.088, -50.246, 106.214, 214.77, 108.084, -179.592, -2414.985]
  MoveL 1105 to (11.76, 312.2, 20) mm, rotated rx -90 ry -25 rz -140.7 deg; joints [-6.709, -50.143, 106.006, 215.007, 108.12, -179.838, -2419.296]
  MoveL 1106 to (6.67, 313.01, 30) mm, rotated rx -90 ry -25 rz -136.04 deg; joints [-6.332, -50.036, 105.793, 215.242, 108.155, -180.085, -2423.955]
  MoveL 1107 to (1.18, 313.37, 40) mm, rotated rx -90 ry -25 rz -131.07 deg; joints [-5.956, -49.924, 105.573, 215.476, 108.19, -180.333, -2428.933]
  MoveL 1108 to (-4.64, 313.2, 50) mm, rotated rx -90 ry -25 rz -125.8 deg; joints [-5.581, -49.807, 105.347, 215.708, 108.224, -180.581, -2434.198]
  MoveL 1109 to (-10.69, 312.41, 60) mm, rotated rx -90 ry -25 rz -120.28 deg; joints [-5.207, -49.684, 105.115, 215.938, 108.259, -180.83, -2439.72]
  MoveL 1110 to (-16.86, 310.92, 70) mm, rotated rx -90 ry -25 rz -114.53 deg; joints [-4.834, -49.556, 104.876, 216.166, 108.295, -181.078, -2445.47]
  MoveL 1111 to (-23.03, 308.7, 80) mm, rotated rx -90 ry -25 rz -108.58 deg; joints [-4.463, -49.423, 104.632, 216.393, 108.331, -181.327, -2451.421]
  MoveL 1112 to (-29.06, 305.72, 90) mm, rotated rx -90 ry -25 rz -102.46 deg; joints [-4.093, -49.283, 104.382, 216.619, 108.368, -181.575, -2457.545]
  MoveL 1113 to (-34.83, 302, 100) mm, rotated rx -90 ry -25 rz -96.19 deg; joints [-3.725, -49.138, 104.126, 216.842, 108.405, -181.823, -2463.814]
  MoveL 1114 to (-40.19, 297.56, 110) mm, rotated rx -90 ry -25 rz -89.8 deg; joints [-3.358, -48.988, 103.864, 217.064, 108.442, -182.072, -2470.201]
  MoveL 1115 to (-45.04, 292.47, 120) mm, rotated rx -90 ry -25 rz -83.32 deg; joints [-2.992, -48.832, 103.595, 217.285, 108.48, -182.32, -2476.68]
  MoveL 1116 to (-49.26, 286.82, 130) mm, rotated rx -90 ry -25 rz -76.78 deg; joints [-2.628, -48.671, 103.321, 217.503, 108.518, -182.569, -2483.221]
  MoveL 1117 to (-52.77, 280.72, 140) mm, rotated rx -90 ry -25 rz -70.2 deg; joints [-2.265, -48.505, 103.04, 217.719, 108.556, -182.819, -2489.796]
  MoveL 1118 to (-55.51, 274.28, 150) mm, rotated rx -90 ry -25 rz -63.63 deg; joints [-1.904, -48.334, 102.753, 217.934, 108.592, -183.069, -2496.375]
  MoveL 1119 to (-57.45, 267.65, 160) mm, rotated rx -90 ry -25 rz -57.07 deg; joints [-1.544, -48.16, 102.46, 218.146, 108.628, -183.32, -2502.926]
  MoveL 1120 to (-58.59, 260.95, 170) mm, rotated rx -90 ry -25 rz -50.58 deg; joints [-1.185, -47.982, 102.161, 218.356, 108.662, -183.573, -2509.416]
  MoveL 1121 to (-58.95, 254.32, 180) mm, rotated rx -90 ry -25 rz -44.19 deg; joints [-0.828, -47.801, 101.855, 218.563, 108.694, -183.828, -2515.809]
  MoveL 1122 to (-58.59, 247.88, 190) mm, rotated rx -90 ry -25 rz -37.93 deg; joints [-0.473, -47.618, 101.543, 218.768, 108.724, -184.086, -2522.068]
  MoveL 1123 to (-57.57, 241.75, 200) mm, rotated rx -90 ry -25 rz -31.84 deg; joints [-0.119, -47.432, 101.224, 218.971, 108.752, -184.345, -2528.155]
  MoveL 1124 to (-56, 236.01, 210) mm, rotated rx -90 ry -25 rz -25.97 deg; joints [0.233, -47.244, 100.899, 219.17, 108.776, -184.608, -2534.028]
  MoveL 1125 to (-53.98, 230.73, 220) mm, rotated rx -90 ry -25 rz -20.35 deg; joints [0.584, -47.055, 100.567, 219.367, 108.797, -184.873, -2539.646]
  MoveL 1126 to (-51.62, 225.97, 230) mm, rotated rx -90 ry -25 rz -15.04 deg; joints [0.933, -46.864, 100.228, 219.56, 108.815, -185.142, -2544.964]
  MoveL 1127 to (-49.06, 221.75, 240) mm, rotated rx -90 ry -25 rz -10.06 deg; joints [1.28, -46.672, 99.883, 219.751, 108.83, -185.414, -2549.94]
  MoveL 1128 to (-46.4, 218.08, 250) mm, rotated rx -90 ry -25 rz -5.47 deg; joints [1.626, -46.479, 99.531, 219.939, 108.841, -185.69, -2554.527]
  MoveL 1129 to (-43.78, 214.95, 260) mm, rotated rx -90 ry -25 rz -1.32 deg; joints [1.97, -46.284, 99.173, 220.123, 108.849, -185.969, -2558.681]
  MoveL 1130 to (-41.29, 212.35, 270) mm, rotated rx -90 ry -25 rz 2.36 deg; joints [2.312, -46.089, 98.807, 220.305, 108.853, -186.252, -2562.358]
  MoveL 1131 to (-39.03, 210.26, 280) mm, rotated rx -90 ry -25 rz 5.51 deg; joints [2.653, -45.891, 98.435, 220.483, 108.854, -186.538, -2565.515]
  MoveL 1132 to (-37.11, 208.63, 290) mm, rotated rx -90 ry -25 rz 8.11 deg; joints [2.992, -45.692, 98.056, 220.659, 108.852, -186.827, -2568.107]
  MoveL 1133 to (-43.85, 188.95, 290) mm, rotated rx -90 ry -25 rz 14.31 deg; joints [2.992, -46.574, 97.966, 220.447, 108.114, -187.494, -2574.314]
  Set speed (60.0 mm/s)
  MoveL 1134 to (-46.6, 190.89, 280) mm, rotated rx -90 ry -25 rz 11.75 deg; joints [2.653, -46.775, 98.344, 220.272, 108.112, -187.203, -2571.748]
  MoveL 1135 to (-49.86, 193.4, 270) mm, rotated rx -90 ry -25 rz 8.62 deg; joints [2.312, -46.974, 98.716, 220.094, 108.107, -186.916, -2568.621]
  MoveL 1136 to (-53.49, 196.56, 260) mm, rotated rx -90 ry -25 rz 4.97 deg; joints [1.97, -47.172, 99.081, 219.913, 108.099, -186.633, -2564.974]
  MoveL 1137 to (-57.36, 200.4, 250) mm, rotated rx -90 ry -25 rz 0.85 deg; joints [1.626, -47.368, 99.44, 219.729, 108.088, -186.352, -2560.848]
  MoveL 1138 to (-61.34, 204.96, 240) mm, rotated rx -90 ry -25 rz -3.71 deg; joints [1.28, -47.563, 99.791, 219.542, 108.074, -186.075, -2556.286]
  MoveL 1139 to (-65.27, 210.27, 230) mm, rotated rx -90 ry -25 rz -8.67 deg; joints [0.933, -47.757, 100.136, 219.352, 108.055, -185.802, -2551.328]
  MoveL 1140 to (-68.98, 216.33, 220) mm, rotated rx -90 ry -25 rz -13.98 deg; joints [0.584, -47.949, 100.474, 219.159, 108.034, -185.532, -2546.018]
  MoveL 1141 to (-72.31, 223.11, 210) mm, rotated rx -90 ry -25 rz -19.6 deg; joints [0.233, -48.14, 100.805, 218.963, 108.008, -185.265, -2540.399]
  MoveL 1142 to (-75.1, 230.56, 200) mm, rotated rx -90 ry -25 rz -25.49 deg; joints [-0.119, -48.329, 101.13, 218.764, 107.98, -185.001, -2534.511]
  MoveL 1143 to (-77.2, 238.6, 190) mm, rotated rx -90 ry -25 rz -31.6 deg; joints [-0.473, -48.517, 101.448, 218.563, 107.948, -184.74, -2528.397]
  MoveL 1144 to (-78.47, 247.13, 180) mm, rotated rx -90 ry -25 rz -37.9 deg; joints [-0.828, -48.703, 101.76, 218.358, 107.914, -184.481, -2522.096]
  MoveL 1145 to (-78.79, 256, 170) mm, rotated rx -90 ry -25 rz -44.35 deg; joints [-1.185, -48.886, 102.065, 218.152, 107.877, -184.226, -2515.648]
  MoveL 1146 to (-78.09, 265.05, 160) mm, rotated rx -90 ry -25 rz -50.91 deg; joints [-1.544, -49.066, 102.363, 217.942, 107.838, -183.972, -2509.09]
  MoveL 1147 to (-76.31, 274.12, 150) mm, rotated rx -90 ry -25 rz -57.54 deg; joints [-1.904, -49.244, 102.656, 217.731, 107.797, -183.719, -2502.46]
  MoveL 1148 to (-73.44, 283.02, 140) mm, rotated rx -90 ry -25 rz -64.21 deg; joints [-2.265, -49.417, 102.942, 217.517, 107.754, -183.468, -2495.79]
  MoveL 1149 to (-69.5, 291.57, 130) mm, rotated rx -90 ry -25 rz -70.88 deg; joints [-2.628, -49.587, 103.221, 217.301, 107.711, -183.218, -2489.115]
  MoveL 1150 to (-64.57, 299.61, 120) mm, rotated rx -90 ry -25 rz -77.53 deg; joints [-2.992, -49.751, 103.495, 217.083, 107.667, -182.969, -2482.468]
  MoveL 1151 to (-58.74, 306.97, 110) mm, rotated rx -90 ry -25 rz -84.12 deg; joints [-3.358, -49.911, 103.762, 216.864, 107.624, -182.72, -2475.878]
  MoveL 1152 to (-52.14, 313.53, 100) mm, rotated rx -90 ry -25 rz -90.62 deg; joints [-3.725, -50.066, 104.024, 216.642, 107.58, -182.471, -2469.376]
  MoveL 1153 to (-44.91, 319.19, 90) mm, rotated rx -90 ry -25 rz -97.01 deg; joints [-4.093, -50.215, 104.279, 216.419, 107.536, -182.222, -2462.991]
  MoveL 1154 to (-37.24, 323.88, 80) mm, rotated rx -90 ry -25 rz -103.25 deg; joints [-4.463, -50.358, 104.529, 216.195, 107.494, -181.973, -2456.752]
  MoveL 1155 to (-29.3, 327.59, 70) mm, rotated rx -90 ry -25 rz -109.31 deg; joints [-4.834, -50.496, 104.772, 215.968, 107.451, -181.724, -2450.689]
  MoveL 1156 to (-21.27, 330.31, 60) mm, rotated rx -90 ry -25 rz -115.17 deg; joints [-5.207, -50.628, 105.01, 215.74, 107.41, -181.474, -2444.831]
  MoveL 1157 to (-13.31, 332.11, 50) mm, rotated rx -90 ry -25 rz -120.79 deg; joints [-5.581, -50.755, 105.242, 215.511, 107.369, -181.225, -2439.206]
  MoveL 1158 to (-5.58, 333.04, 40) mm, rotated rx -90 ry -25 rz -126.15 deg; joints [-5.956, -50.876, 105.467, 215.28, 107.328, -180.976, -2433.845]
  MoveL 1159 to (1.77, 333.22, 30) mm, rotated rx -90 ry -25 rz -131.22 deg; joints [-6.332, -50.991, 105.687, 215.047, 107.287, -180.727, -2428.779]
  MoveL 1160 to (8.64, 332.76, 20) mm, rotated rx -90 ry -25 rz -135.96 deg; joints [-6.709, -51.103, 105.901, 214.813, 107.247, -180.478, -2424.039]
  MoveL 1161 to (14.93, 331.81, 10) mm, rotated rx -90 ry -25 rz -140.34 deg; joints [-7.088, -51.209, 106.109, 214.576, 107.206, -180.23, -2419.656]
  MoveL 1162 to (20.57, 330.51, 0) mm, rotated rx -90 ry -25 rz -144.34 deg; joints [-7.468, -51.311, 106.31, 214.338, 107.164, -179.983, -2415.665]
  MoveL 1163 to (-43.85, 188.95, 290) mm, rotated rx -90 ry -25 rz 14.31 deg; joints [2.992, -46.574, 97.966, 220.447, 108.114, -187.494, -2574.314]
  Set speed (60.0 mm/s)
  MoveL 1164 to (-28.22, 202.67, 290) mm, rotated rx -90 ry -25 rz 19.2 deg; joints [2.992, -45.67, 98.058, 220.664, 108.87, -186.811, -2579.196]
  MoveL 1165 to (20.57, 330.51, 0) mm, rotated rx -90 ry -25 rz -144.34 deg; joints [-7.468, -51.311, 106.31, 214.338, 107.164, -179.983, -2415.665]
  Set speed (60.0 mm/s)
  MoveL 1166 to (10.16, 312.5, 0) mm, rotated rx -90 ry -25 rz -139.23 deg; joints [-7.468, -50.355, 106.415, 214.529, 108.039, -179.354, -2420.767]
  MoveL 1167 to (20.57, 330.51, 0) mm, rotated rx -90 ry -25 rz -144.34 deg; joints [-7.468, -51.311, 106.31, 214.338, 107.164, -179.983, -2415.665]
  Set speed (60.0 mm/s)
  MoveL 1168 to (14.93, 331.81, 10) mm, rotated rx -90 ry -25 rz -140.34 deg; joints [-7.088, -51.209, 106.109, 214.576, 107.206, -180.23, -2419.656]
  MoveL 1169 to (8.64, 332.76, 20) mm, rotated rx -90 ry -25 rz -135.96 deg; joints [-6.709, -51.103, 105.901, 214.813, 107.247, -180.478, -2424.039]
  MoveL 1170 to (1.77, 333.22, 30) mm, rotated rx -90 ry -25 rz -131.22 deg; joints [-6.332, -50.991, 105.687, 215.047, 107.287, -180.727, -2428.779]
  MoveL 1171 to (-5.58, 333.04, 40) mm, rotated rx -90 ry -25 rz -126.15 deg; joints [-5.956, -50.876, 105.467, 215.28, 107.328, -180.976, -2433.845]
  MoveL 1172 to (-13.31, 332.11, 50) mm, rotated rx -90 ry -25 rz -120.79 deg; joints [-5.581, -50.755, 105.242, 215.511, 107.369, -181.225, -2439.206]
  MoveL 1173 to (-21.27, 330.31, 60) mm, rotated rx -90 ry -25 rz -115.17 deg; joints [-5.207, -50.628, 105.01, 215.74, 107.41, -181.474, -2444.831]
  MoveL 1174 to (-29.3, 327.59, 70) mm, rotated rx -90 ry -25 rz -109.31 deg; joints [-4.834, -50.496, 104.772, 215.968, 107.451, -181.724, -2450.689]
  MoveL 1175 to (-37.24, 323.88, 80) mm, rotated rx -90 ry -25 rz -103.25 deg; joints [-4.463, -50.358, 104.529, 216.195, 107.494, -181.973, -2456.752]
  MoveL 1176 to (-44.91, 319.19, 90) mm, rotated rx -90 ry -25 rz -97.01 deg; joints [-4.093, -50.215, 104.279, 216.419, 107.536, -182.222, -2462.991]
  MoveL 1177 to (-52.14, 313.53, 100) mm, rotated rx -90 ry -25 rz -90.62 deg; joints [-3.725, -50.066, 104.024, 216.642, 107.58, -182.471, -2469.376]
  MoveL 1178 to (-58.74, 306.97, 110) mm, rotated rx -90 ry -25 rz -84.12 deg; joints [-3.358, -49.911, 103.762, 216.864, 107.624, -182.72, -2475.878]
  MoveL 1179 to (-64.57, 299.61, 120) mm, rotated rx -90 ry -25 rz -77.53 deg; joints [-2.992, -49.751, 103.495, 217.083, 107.667, -182.969, -2482.468]
  MoveL 1180 to (-69.5, 291.57, 130) mm, rotated rx -90 ry -25 rz -70.88 deg; joints [-2.628, -49.587, 103.221, 217.301, 107.711, -183.218, -2489.115]
  MoveL 1181 to (-73.44, 283.02, 140) mm, rotated rx -90 ry -25 rz -64.21 deg; joints [-2.265, -49.417, 102.942, 217.517, 107.754, -183.468, -2495.79]
  MoveL 1182 to (-76.31, 274.12, 150) mm, rotated rx -90 ry -25 rz -57.54 deg; joints [-1.904, -49.244, 102.656, 217.731, 107.797, -183.719, -2502.46]
  MoveL 1183 to (-78.09, 265.05, 160) mm, rotated rx -90 ry -25 rz -50.91 deg; joints [-1.544, -49.066, 102.363, 217.942, 107.838, -183.972, -2509.09]
  MoveL 1184 to (-78.79, 256, 170) mm, rotated rx -90 ry -25 rz -44.35 deg; joints [-1.185, -48.886, 102.065, 218.152, 107.877, -184.226, -2515.648]
  MoveL 1185 to (-78.47, 247.13, 180) mm, rotated rx -90 ry -25 rz -37.9 deg; joints [-0.828, -48.703, 101.76, 218.358, 107.914, -184.481, -2522.096]
  MoveL 1186 to (-77.2, 238.6, 190) mm, rotated rx -90 ry -25 rz -31.6 deg; joints [-0.473, -48.517, 101.448, 218.563, 107.948, -184.74, -2528.397]
  MoveL 1187 to (-75.1, 230.56, 200) mm, rotated rx -90 ry -25 rz -25.49 deg; joints [-0.119, -48.329, 101.13, 218.764, 107.98, -185.001, -2534.511]
  MoveL 1188 to (-72.31, 223.11, 210) mm, rotated rx -90 ry -25 rz -19.6 deg; joints [0.233, -48.14, 100.805, 218.963, 108.008, -185.265, -2540.399]
  MoveL 1189 to (-68.98, 216.33, 220) mm, rotated rx -90 ry -25 rz -13.98 deg; joints [0.584, -47.949, 100.474, 219.159, 108.034, -185.532, -2546.018]
  MoveL 1190 to (-65.27, 210.27, 230) mm, rotated rx -90 ry -25 rz -8.67 deg; joints [0.933, -47.757, 100.136, 219.352, 108.055, -185.802, -2551.328]
  MoveL 1191 to (-61.34, 204.96, 240) mm, rotated rx -90 ry -25 rz -3.71 deg; joints [1.28, -47.563, 99.791, 219.542, 108.074, -186.075, -2556.286]
  MoveL 1192 to (-57.36, 200.4, 250) mm, rotated rx -90 ry -25 rz 0.85 deg; joints [1.626, -47.368, 99.44, 219.729, 108.088, -186.352, -2560.848]
  MoveL 1193 to (-53.49, 196.56, 260) mm, rotated rx -90 ry -25 rz 4.97 deg; joints [1.97, -47.172, 99.081, 219.913, 108.099, -186.633, -2564.974]
  MoveL 1194 to (-49.86, 193.4, 270) mm, rotated rx -90 ry -25 rz 8.62 deg; joints [2.312, -46.974, 98.716, 220.094, 108.107, -186.916, -2568.621]
  MoveL 1195 to (-46.6, 190.89, 280) mm, rotated rx -90 ry -25 rz 11.75 deg; joints [2.653, -46.775, 98.344, 220.272, 108.112, -187.203, -2571.748]
  MoveL 1196 to (-43.85, 188.95, 290) mm, rotated rx -90 ry -25 rz 14.31 deg; joints [2.992, -46.574, 97.966, 220.447, 108.114, -187.494, -2574.314]
  MoveL 1197 to (-28.22, 202.67, 290) mm, rotated rx -90 ry -25 rz 19.2 deg; joints [2.992, -45.67, 98.058, 220.664, 108.87, -186.811, -2579.196]
  Set speed (60.0 mm/s)
  MoveL 1198 to (-30.4, 203.93, 280) mm, rotated rx -90 ry -25 rz 16.58 deg; joints [2.653, -45.868, 98.437, 220.489, 108.873, -186.521, -2576.579]
  MoveL 1199 to (-33, 205.58, 270) mm, rotated rx -90 ry -25 rz 13.39 deg; joints [2.312, -46.064, 98.809, 220.311, 108.874, -186.234, -2573.391]
  MoveL 1200 to (-35.92, 207.69, 260) mm, rotated rx -90 ry -25 rz 9.67 deg; joints [1.97, -46.258, 99.175, 220.13, 108.871, -185.95, -2569.674]
  MoveL 1201 to (-39.07, 210.28, 250) mm, rotated rx -90 ry -25 rz 5.47 deg; joints [1.626, -46.451, 99.533, 219.946, 108.865, -185.669, -2565.473]
  MoveL 1202 to (-42.34, 213.41, 240) mm, rotated rx -90 ry -25 rz 0.83 deg; joints [1.28, -46.642, 99.885, 219.758, 108.855, -185.392, -2560.831]
  MoveL 1203 to (-45.62, 217.1, 230) mm, rotated rx -90 ry -25 rz -4.21 deg; joints [0.933, -46.832, 100.231, 219.568, 108.842, -185.119, -2555.794]
  MoveL 1204 to (-48.8, 221.36, 220) mm, rotated rx -90 ry -25 rz -9.59 deg; joints [0.584, -47.021, 100.57, 219.375, 108.826, -184.849, -2550.406]
  MoveL 1205 to (-51.74, 226.19, 210) mm, rotated rx -90 ry -25 rz -15.29 deg; joints [0.233, -47.209, 100.902, 219.178, 108.806, -184.582, -2544.713]
  MoveL 1206 to (-54.33, 231.55, 200) mm, rotated rx -90 ry -25 rz -21.24 deg; joints [-0.119, -47.395, 101.227, 218.979, 108.783, -184.319, -2538.758]
  MoveL 1207 to (-56.44, 237.4, 190) mm, rotated rx -90 ry -25 rz -27.41 deg; joints [-0.473, -47.58, 101.546, 218.777, 108.756, -184.059, -2532.587]
  MoveL 1208 to (-57.96, 243.66, 180) mm, rotated rx -90 ry -25 rz -33.76 deg; joints [-0.828, -47.763, 101.858, 218.572, 108.727, -183.801, -2526.24]
  MoveL 1209 to (-58.8, 250.25, 170) mm, rotated rx -90 ry -25 rz -40.24 deg; joints [-1.185, -47.944, 102.164, 218.365, 108.694, -183.547, -2519.76]
  MoveL 1210 to (-58.89, 257.04, 160) mm, rotated rx -90 ry -25 rz -46.82 deg; joints [-1.544, -48.123, 102.464, 218.154, 108.66, -183.294, -2513.183]
  MoveL 1211 to (-58.18, 263.92, 150) mm, rotated rx -90 ry -25 rz -53.45 deg; joints [-1.904, -48.298, 102.757, 217.942, 108.623, -183.043, -2506.549]
  MoveL 1212 to (-56.65, 270.74, 140) mm, rotated rx -90 ry -25 rz -60.11 deg; joints [-2.265, -48.47, 103.043, 217.727, 108.585, -182.794, -2499.89]
  MoveL 1213 to (-54.3, 277.38, 130) mm, rotated rx -90 ry -25 rz -66.76 deg; joints [-2.628, -48.638, 103.324, 217.51, 108.546, -182.546, -2493.241]
  MoveL 1214 to (-51.17, 283.7, 120) mm, rotated rx -90 ry -25 rz -73.37 deg; joints [-2.992, -48.802, 103.598, 217.291, 108.506, -182.299, -2486.632]
  MoveL 1215 to (-47.33, 289.58, 110) mm, rotated rx -90 ry -25 rz -79.91 deg; joints [-3.358, -48.961, 103.866, 217.07, 108.466, -182.053, -2480.094]
  MoveL 1216 to (-42.85, 294.92, 100) mm, rotated rx -90 ry -25 rz -86.35 deg; joints [-3.725, -49.114, 104.128, 216.848, 108.426, -181.807, -2473.654]
  MoveL 1217 to (-37.86, 299.62, 90) mm, rotated rx -90 ry -25 rz -92.66 deg; joints [-4.093, -49.263, 104.384, 216.623, 108.386, -181.561, -2467.341]
  MoveL 1218 to (-32.46, 303.64, 80) mm, rotated rx -90 ry -25 rz -98.82 deg; joints [-4.463, -49.406, 104.634, 216.397, 108.346, -181.315, -2461.181]
  MoveL 1219 to (-26.8, 306.94, 70) mm, rotated rx -90 ry -25 rz -104.8 deg; joints [-4.834, -49.543, 104.878, 216.169, 108.307, -181.069, -2455.202]
  MoveL 1220 to (-21, 309.52, 60) mm, rotated rx -90 ry -25 rz -110.57 deg; joints [-5.207, -49.675, 105.115, 215.94, 108.268, -180.823, -2449.431]
  MoveL 1221 to (-15.19, 311.39, 50) mm, rotated rx -90 ry -25 rz -116.1 deg; joints [-5.581, -49.801, 105.347, 215.709, 108.23, -180.577, -2443.896]
  MoveL 1222 to (-9.5, 312.61, 40) mm, rotated rx -90 ry -25 rz -121.38 deg; joints [-5.956, -49.921, 105.573, 215.476, 108.192, -180.331, -2438.624]
  MoveL 1223 to (-4.03, 313.25, 30) mm, rotated rx -90 ry -25 rz -126.35 deg; joints [-6.332, -50.037, 105.793, 215.242, 108.154, -180.086, -2433.645]
  MoveL 1224 to (1.12, 313.37, 20) mm, rotated rx -90 ry -25 rz -131.01 deg; joints [-6.709, -50.147, 106.006, 215.006, 108.116, -179.841, -2428.989]
  MoveL 1225 to (5.87, 313.09, 10) mm, rotated rx -90 ry -25 rz -135.31 deg; joints [-7.088, -50.253, 106.214, 214.768, 108.078, -179.597, -2424.685]
  MoveL 1226 to (10.16, 312.5, 0) mm, rotated rx -90 ry -25 rz -139.23 deg; joints [-7.468, -50.355, 106.415, 214.529, 108.039, -179.354, -2420.767]
  Set speed (1000.0 mm/s)
  MoveL 1227 to (10.16, 312.5, 0) mm, rotated rx -90 ry -25 rz -139.23 deg; joints [-7.468, -50.355, 106.415, 214.529, 108.039, -179.354, -2420.767]
